(* PLC project KA107__GPA2.project, Prosoft-Systems Ltd. Astra.IDE Astra.IDE_V1.7.2.1 *)
(* stored: creationDateTime 2025-08-26T12:04:32.1909898, modificationDateTime 2025-08-26T12:03:09.7987139 *)

///
///Назначение: 		готовности к пуску
///Автор: 				Korsuntsev/Chekmarev 20/02/2025
///Версия: 			00.00.02
///Проект: 			КА107
{attribute 'qualified_only' := ''}
{attribute 'strict' := ''}
{attribute 'symbol' := 'none'}
TYPE ENUM_ReadyToStart :
(
	/// Готовность отключена
	OFF := 0,
	/// Готовность к ХП
	HP := 1,
	/// Готовность к КПК
	KPK := 2,
	/// Готовность к АПК
	APK := 3
) USINT;
END_TYPE

PROGRAM DIAGN

                    REDUNDANCY();
UCP1_A1_1();
UCP1_A2_1();
UE1_A1_1();

                  

ACTION UE1_A1_1:
                        PsDiagn.PROXY_ST_XX_X1X(MODULE := UE1_A1_ST1, DATA := MODULE_UE1_A1_ST1);
PsDiagn.PROXY_PP_00_XXX(MODULE := UE1_A1_PP1, DATA := MODULE_UE1_A1_PP1);
PsDiagn.PROXY_AI_16_011(MODULE := UE1_A1_DI1, DATA := MODULE_UE1_A1_DI1);
PsDiagn.PROXY_AI_16_011(MODULE := UE1_A1_DI2, DATA := MODULE_UE1_A1_DI2);
PsDiagn.PROXY_AI_16_011(MODULE := UE1_A1_DI3, DATA := MODULE_UE1_A1_DI3);
PsDiagn.PROXY_DI_32_011(MODULE := UE1_A1_DI4, DATA := MODULE_UE1_A1_DI4);
PsDiagn.PROXY_DI_32_011(MODULE := UE1_A1_DI5, DATA := MODULE_UE1_A1_DI5);
PsDiagn.PROXY_DO_32_012(MODULE := UE1_A1_DO1, DATA := MODULE_UE1_A1_DO1);
PsDiagn.PROXY_DI_32_011(MODULE := UE1_A1_DI6, DATA := MODULE_UE1_A1_DI6);
PsDiagn.PROXY_DO_32_012(MODULE := UE1_A1_DO2, DATA := MODULE_UE1_A1_DO2);
PsDiagn.PROXY_DI_32_011(MODULE := UE1_A1_DI7, DATA := MODULE_UE1_A1_DI7);
PsDiagn.PROXY_ST_XX_X2X(MODULE := UE1_A1_ST2, DATA := MODULE_UE1_A1_ST2);

                      
END_ACTION

ACTION UCP1_A2_1:
                        PsDiagn.PROXY_ST_XX_X1X(MODULE := UCP1_A2_ST1, DATA := MODULE_UCP1_A2_ST1);
PsDiagn.PROXY_PP_00_XXX(MODULE := UCP1_A2_PP1, DATA := MODULE_UCP1_A2_PP1);
PsDiagn.PROXY_AO_08_031(MODULE := UCP1_A2_AO1, DATA := MODULE_UCP1_A2_AO1);
PsDiagn.PROXY_AI_16_011(MODULE := UCP1_A2_DI1, DATA := MODULE_UCP1_A2_DI1);
PsDiagn.PROXY_AI_16_011(MODULE := UCP1_A2_DI2, DATA := MODULE_UCP1_A2_DI2);
PsDiagn.PROXY_DI_32_011(MODULE := UCP1_A2_DI3, DATA := MODULE_UCP1_A2_DI3);
PsDiagn.PROXY_DO_32_012(MODULE := UCP1_A2_DO1, DATA := MODULE_UCP1_A2_DO1);
PsDiagn.PROXY_DI_32_011(MODULE := UCP1_A2_DI4, DATA := MODULE_UCP1_A2_DI4);
PsDiagn.PROXY_ST_XX_X2X(MODULE := UCP1_A2_ST2, DATA := MODULE_UCP1_A2_ST2);

                      
END_ACTION

ACTION REDUNDANCY:
                        //Активный ПЛК
IS_ACTIVE := TRUE;

//ПЛК А
IS_CPU_A := TRUE;

//ПЛК В
IS_CPU_B := FALSE;


                      
END_ACTION

ACTION UCP1_A1_1:
                        PsDiagn.PROXY_ST_XX_X1X(MODULE := UCP1_A1_ST1, DATA := MODULE_UCP1_A1_ST1);
PsDiagn.PROXY_PP_00_XXX(MODULE := UCP1_A1_PP1, DATA := MODULE_UCP1_A1_PP1);
PsDiagn.GET_CPU_INFO_R500(REGULBUS_HW := Regul_Bus_OS.HwError, SYNC_OK := TRUE, HW := UCP1_A1_CU1.HwError, PF := FALSE, INFO => MODULE_UCP1_A1_CU1);
PsDiagn.PROXY_DA_03_021_L_FRQ(MODULE := UCP1_A1_FI1, DATA := MODULE_UCP1_A1_FI1);
PsDiagn.PROXY_DA_03_021_L_FRQ(MODULE := UCP1_A1_FI2, DATA := MODULE_UCP1_A1_FI2);
PsDiagn.PROXY_AI_08_052(MODULE := UCP1_A1_AI1, DATA := MODULE_UCP1_A1_AI1);
PsDiagn.PROXY_AI_08_052(MODULE := UCP1_A1_AI2, DATA := MODULE_UCP1_A1_AI2);
PsDiagn.PROXY_AI_08_052(MODULE := UCP1_A1_AI3, DATA := MODULE_UCP1_A1_AI3);
PsDiagn.PROXY_AI_08_031(MODULE := UCP1_A1_AI4, DATA := MODULE_UCP1_A1_AI4);
PsDiagn.PROXY_AI_08_031(MODULE := UCP1_A1_AI5, DATA := MODULE_UCP1_A1_AI5);
PsDiagn.PROXY_AI_08_031(MODULE := UCP1_A1_AI6, DATA := MODULE_UCP1_A1_AI6);
PsDiagn.PROXY_AI_08_031(MODULE := UCP1_A1_AI7, DATA := MODULE_UCP1_A1_AI7);
PsDiagn.PROXY_ST_XX_X2X(MODULE := UCP1_A1_ST2, DATA := MODULE_UCP1_A1_ST2);

                      
END_ACTION
END_PROGRAM

FUNCTION FC_PrepareShutdown : DWORD
VAR_IN_OUT
	EventPrm: Component_Manager.EVTPARAM_CmpMgr_Shutdown;
END_VAR
VAR
END_VAR

                    IS_ACTIVE := FALSE;
IS_CPU_A := FALSE;
IS_CPU_B := FALSE;

                  
END_FUNCTION

FUNCTION FC_StopDone : DWORD
VAR_IN_OUT
	EventPrm: CmpApp.EVTPARAM_CmpAppStop;
END_VAR
VAR
END_VAR

                    IS_ACTIVE := FALSE;
IS_CPU_A := FALSE;
IS_CPU_B := FALSE;

                  
END_FUNCTION

FUNCTION FC_Exception : DWORD
VAR_IN_OUT
	EventPrm: CmpApp.EVTPARAM_CmpAppException;
END_VAR
VAR
END_VAR

                    IS_ACTIVE := FALSE;
IS_CPU_A := FALSE;
IS_CPU_B := FALSE;

                  
END_FUNCTION

{attribute 'linkalways' := ''}
PROGRAM PRG_9d6fa412_87bb_44d3_b4af_3b2a0d18f6a8

                    {IF defined (pou: SETPOINTS_PRG_STORE_060ed6ea_c6b5_480d_b15e_3bc8654c83ea)}
SETPOINTS_PRG_STORE_060ed6ea_c6b5_480d_b15e_3bc8654c83ea();
{END_IF}
                  
END_PROGRAM

{attribute 'linkalways' := ''}
PROGRAM PRG_b5ed8c35_93f2_4693_9ede_6cbb2df9f327

                    {IF defined (pou: SETPOINTS_PRG_RESTORE_926b34b1_d125_4ae4_9712_933a3ae333bd)}
SETPOINTS_PRG_RESTORE_926b34b1_d125_4ae4_9712_933a3ae333bd();
{END_IF}
                  
END_PROGRAM

PROGRAM PRG_base
VAR
 	//Время выполнения программы
	result_time:ULINT;
	/// Признак первого вызова программы
	init: BOOL := TRUE;
END_VAR
VAR_TEMP
	start_time:ULINT;
	end_time:ULINT;
END_VAR

                    start_time:= PsTimeGetUtcTimeNs(); // Время начала выполнения
//==============================================================================================

IF init THEN
	fun_init();
	init := FALSE;
END_IF

//Кнопки
btn_update();

// Настройки
tunpar_update();

// Таймеры
tmr_update();

// ИМ-ы
// Конфигуратор
am_update();
// Создан вручную
am_update_base();

//Алгоритм
ALG_base();				//Алгоритм

aggregation_am();

// Формирование тестовых сигналов
test.Saw_Slow();
test.Sin_Slow();

//==============================================================================================
end_time:=PsTimeGetUtcTimeNs() ;  // конец
result_time:=end_time-start_time;  // время выполнения фрагмента кода
                  
END_PROGRAM

PROGRAM PRG_fast
VAR
 	//Время выполнения программы
	result_time:ULINT;
END_VAR
VAR_TEMP
	start_time:ULINT;
	end_time:ULINT;
END_VAR

                    start_time:=PsTimeGetUtcTimeNs(); // Время начала выполнения
//==============================================================================================

////// Временно здесь
//{warning ' Убрать на новой версии макроса '}
//aipar.common.sim_aggregated	:= FALSE;
//aopar.common.sim_aggregated	:= FALSE;
//dipar.common.sim_aggregated	:= FALSE;
//dopar.common.sim_aggregated	:= FALSE;
/////////////

// Сброс переменных VAR_STAT
// По входам / выходам
reset_io_var_stat();
// По сигнализациям
reset_alarm_var_stat();
// По ИМам
reset_am_var_stat();

// Ввод
	aipar_update(cycle := cycle_time_fast);		//Вызов обработки всех экземпляров AI быстрого цикла
	dipar_update();								//Вызов обработки всех экземпляров DI быстрого цикла
	
	MODULE_UCP1_A1_AI6.T_JUNCTION := aipar.Tcool.value; // компенсация холодного спая
	MODULE_UCP1_A1_AI7.T_JUNCTION := aipar.Tcool.value; // компенсация холодного спая
//---------------------------------------------------------------------------------------------

// Расчётные параметры
	acpar_handler.handler(cycle := cycle_time_fast);
	
	acpar_update(); 							//Обработка расчётных параметров (Формирование уставок)
//---------------------------------------------------------------------------------------------	

// Сигнализации
	Alarm_link(); //Подготовка данных и вызов обработчиков сигнализаций
//Агрегация сигнализаций (все сигнализации должны быть вызваны к этому моменту)
	aggregation_alarms();
//---------------------------------------------------------------------------------------------	

// Топливный регулятор
	FR_link();
	AS_Link();

// Быстрые ИМ-ы
	ALG_D_AM_fast();
	// Создан вручную
	am_update_fast();
	// аналоговые
	// Конфигуратор
	ama_update();

//Сигналы контроллера
	ALG_PLC();

// Вывод
	aopar_update(); 							//Вызов обработки всех экземпляров AO быстрого цикла
	dopar_update(); 							//Вызов обработки всех экземпляров DO быстрого цикла
//---------------------------------------------------------------------------------------------	
// IEC 104

// Формирование тестовых сигналов
	test.Saw_Fast();
// IEC-104
	IEC104_update();

//==============================================================================================
end_time:=PsTimeGetUtcTimeNs() ;  // конец
result_time:=end_time-start_time;  // время выполнения фрагмента кода

                  
END_PROGRAM

PROGRAM PRG_slow

                    handleMotoClock();
alg.sh_cntrl := ShCntrl();
                  
END_PROGRAM

{region INFO}
(*
 Назначение: Используется для вызова предупредительных и ограничительных сигнализаций
 Автор:  /Andrey/ 24.06.2025 16:50:31
 Версия: v00.00.22
 Проект: KA107__GPA2
*)
{endregion}
FUNCTION alr_update : BOOL
VAR_INPUT
END_VAR

                    //==========================================================================

//==========================================================================
//Подсистема: Внешние источники
//--------------------------------------------------------------------------
//Кнопка ЭАО на ПРУ нажата сигнал 1 (НР)
alr.EAO_PRU_1(
in     := dipar.EAO_PRU_1.value,
cmd_on := TRUE, cmd_off  := FALSE);
//--------------------------------------------------------------------------

//Кнопка ЭАО на ПРУ нажата сигнал 2 (НЗ)
alr.EAO_PRU_2(
in     := dipar.EAO_PRU_2.value,
cmd_on := TRUE, cmd_off  := FALSE);
//--------------------------------------------------------------------------

//Кнопка ЭАО на ПРУ нажата сигнал 3 (НЗ)
alr.EAO_PRU_3(
in     := dipar.EAO_PRU_3.value,
cmd_on := TRUE, cmd_off  := FALSE);
//--------------------------------------------------------------------------

//Нет связи с ПРУ
alr.PRU_noLink(
in     := NOT PRU.Link,
cmd_on := TRUE, cmd_off  := FALSE);
//--------------------------------------------------------------------------

//==========================================================================

//==========================================================================
//Подсистема: Блок двигателя
//--------------------------------------------------------------------------
//Загазованность контейнеров выше нормы
alr.Zagaz_OD_Pv(
in     := dipar.Zagaz_OD_Pv.value,
cmd_on := TRUE, cmd_off  := FALSE);
//--------------------------------------------------------------------------

//Повышенная вибрация двигателя
alr.Vs_D_Pv(
in     := dipar.Vs_D_Pv.value,
cmd_on := TRUE, cmd_off  := FALSE);
//--------------------------------------------------------------------------

//Повыш. Вибрация ТК
alr.Vstk_H(
in     := aipar.Vstk.setpoint.H,
cmd_on := TRUE, cmd_off  := FALSE);
//--------------------------------------------------------------------------

//Повыш. Вибрация СТ
alr.Vsst_H(
in     := aipar.Vsst.setpoint.H,
cmd_on := TRUE, cmd_off  := FALSE);
//--------------------------------------------------------------------------

//Сигнализатор обледенения
alr.Ace_alr(
in     := dipar.Ace_alr.value,
cmd_on := TRUE, cmd_off  := FALSE);
//--------------------------------------------------------------------------

//КПВ не открыты на пуске
alr.KPV_nOpen(
in     := NOT ( dipar.KPV2_ON.value AND dipar.KPV3_ON.value AND dipar.KPV4_ON.value AND dipar.KPV1_ON.value AND dipar.KPV5_ON.value ),
cmd_on := acpar.Ntk.value > 2000 AND acpar.Ntk.value < 4500 AND alg.start, cmd_off  := acpar.Ntk.value > 4500 OR alg.AO);
//--------------------------------------------------------------------------

//КПВ234 не открыты
alr.KPV234_nOpen(
in     := NOT ( dipar.KPV2_ON.value AND dipar.KPV3_ON.value AND dipar.KPV4_ON.value ),
cmd_on := NOss.cmd_KPV234_On OR NObs.cmd_KPV234_On OR AOss.cmd_KPV234_On OR AObs.cmd_KPV234_On, cmd_off  := acpar.Ntk.value < 2000);
//--------------------------------------------------------------------------

//Повыш. Обороты СТ > 8500 об/мин
alr.Nst_H(
in     := acpar.Nst.setpoint.H,
cmd_on := TRUE, cmd_off  := FALSE);
//--------------------------------------------------------------------------

//Высокая скорость изменения оборотов 1-ого канала ТК
alr.Ntk_1_OV(
in     := acpar_handler.handler.nTKcalc.fltUcv[1],
cmd_on := TRUE, cmd_off  := FALSE);
//--------------------------------------------------------------------------

//Высокая скорость изменения оборотов 2-ого канала ТК
alr.Ntk_2_OV(
in     := acpar_handler.handler.nTKcalc.fltUcv[2],
cmd_on := TRUE, cmd_off  := FALSE);
//--------------------------------------------------------------------------

//Значения оборотов 1-ого канала ТК не в диапазоне
alr.Ntk_1_UV(
in     := acpar_handler.handler.nTKcalc.flt[1],
cmd_on := TRUE, cmd_off  := FALSE);
//--------------------------------------------------------------------------

//Значения оборотов 2-ого канала ТК не в диапазоне
alr.Ntk_2_UV(
in     := acpar_handler.handler.nTKcalc.flt[2],
cmd_on := TRUE, cmd_off  := FALSE);
//--------------------------------------------------------------------------

//Значения оборотов 1-ого канала СТ не в диапазоне
alr.Nst_1_UV(
in     := acpar_handler.handler.nSTcalc.flt[1],
cmd_on := TRUE, cmd_off  := FALSE);
//--------------------------------------------------------------------------

//Значения оборотов 2-ого канала СТ не в диапазоне
alr.Nst_2_UV(
in     := acpar_handler.handler.nSTcalc.flt[2],
cmd_on := TRUE, cmd_off  := FALSE);
//--------------------------------------------------------------------------

//Высокая скорость изменения оборотов 1-ого канала СТ
alr.Nst_1_OV(
in     := acpar_handler.handler.nSTcalc.fltUcv[1],
cmd_on := TRUE, cmd_off  := FALSE);
//--------------------------------------------------------------------------

//Высокая скорость изменения оборотов 2-ого канала СТ
alr.Nst_2_OV(
in     := acpar_handler.handler.nSTcalc.fltUcv[2],
cmd_on := TRUE, cmd_off  := FALSE);
//--------------------------------------------------------------------------

//Повыш. Температура газа на входе СТ
alr.Tg_inST_H(
in     := acpar.Tg_inST.setpoint.H,
cmd_on := TRUE, cmd_off  := FALSE);
//--------------------------------------------------------------------------

//Нет сигнала: ТРК: готовность
alr.N_TRKready(
in     := NOT dipar.TRKready.value,
cmd_on := TRUE, cmd_off  := FALSE);
//--------------------------------------------------------------------------

//ТРК: авария
alr.TRKalr(
in     := dipar.TRKalr.value,
cmd_on := TRUE, cmd_off  := FALSE);
//--------------------------------------------------------------------------

//Контроль САУ не пройден
alr.nCheckSAU(
in     := check.tmrCancelPrm.Q,
cmd_on := TRUE, cmd_off  := FALSE);
//--------------------------------------------------------------------------

//Неисправность БЗА
alr.BZA_flt(
in     := NOT dipar.BZA_ready_1.value OR NOT dipar.BZA_ready_2.value,
cmd_on := tch.GTDWork.value, cmd_off  := NOT tch.GTDWork.value);
//--------------------------------------------------------------------------

//==========================================================================

//==========================================================================
//Подсистема: Маслосистема двигателя
//--------------------------------------------------------------------------
//Пониж. Температура масла на входе двигателя
alr.Tm_inD_L(
in     := aipar.Tm_inD.setpoint.L,
cmd_on := TRUE, cmd_off  := FALSE);
//--------------------------------------------------------------------------

//Уровень масла в МБД+Н минимальный
alr.Lm_MB_Pn(
in     := dipar.Lm_MB_Pn.value,
cmd_on := TRUE, cmd_off  := FALSE);
//--------------------------------------------------------------------------

//==========================================================================

//==========================================================================
//Подсистема: Воздушный стартер
//--------------------------------------------------------------------------
//==========================================================================

//==========================================================================
//Подсистема: Аппарат воздушного охлаждения масла двигателя
//--------------------------------------------------------------------------
//Повыш. Температура масла на выходе АВОМД
alr.Tm_outAVOM_H(
in     := aipar.Tm_outAVOM.setpoint.H,
cmd_on := TRUE, cmd_off  := FALSE);
//--------------------------------------------------------------------------

//Неисправность вентилятора 1 АВОМД
alr.Vn1_AVOM_flt(
in     := am.Vn1_AVOM.flt,
cmd_on := TRUE, cmd_off  := FALSE);
//--------------------------------------------------------------------------

//Неисправность вентилятора 2 АВОМД
alr.Vn2_AVOM_flt(
in     := am.Vn2_AVOM.flt,
cmd_on := TRUE, cmd_off  := FALSE);
//--------------------------------------------------------------------------

//Неисправность вентилятора 3 АВОМД
alr.Vn3_AVOM_flt(
in     := am.Vn3_AVOM.flt,
cmd_on := TRUE, cmd_off  := FALSE);
//--------------------------------------------------------------------------

//Неисправность вентилятора 4 АВОМД
alr.Vn4_AVOM_flt(
in     := am.Vn4_AVOM.flt,
cmd_on := TRUE, cmd_off  := FALSE);
//--------------------------------------------------------------------------

//==========================================================================

//==========================================================================
//Подсистема: Блок топливного газа
//--------------------------------------------------------------------------
//Пониж. Давление топливного газа перед ТРК
alr.Ptg_inTRK_L(
in     := aipar.Ptg_inTRK.setpoint.L,
cmd_on := alg.sh_TG, cmd_off  := NOT alg.sh_TG);
//--------------------------------------------------------------------------

//Повыш. Давление топливного газа перед ТРК
alr.Ptg_inTRK_H(
in     := aipar.Ptg_inTRK.setpoint.H,
cmd_on := true, cmd_off  := false);
//--------------------------------------------------------------------------

//Давление газа перед дозатором газа Предупредительное
alr.Ptg_inDG_Pn(
in     := dipar.Ptg_inDG_Pn.value,
cmd_on := alg.sh_TG, cmd_off  := NOT alg.sh_TG);
//--------------------------------------------------------------------------

//==========================================================================

//==========================================================================
//Подсистема: Блок пускового газа
//--------------------------------------------------------------------------
//==========================================================================

//==========================================================================
//Подсистема: Противообледенительная система и воздухоочистное устройство
//--------------------------------------------------------------------------
//Перепад на сетке ВОУ
alr.Exh_VOU(
in     := dipar.Exh_VOU.value,
cmd_on := TRUE, cmd_off  := FALSE);
//--------------------------------------------------------------------------

//==========================================================================

//==========================================================================
//Подсистема: Компрессорная установка/блок нагнетателя
//--------------------------------------------------------------------------
//Опасность помпажа нагнетателя
alr.AS_Pv(
in     := s_tunpar.ASprot.emergOpenBypass,
cmd_on := TRUE, cmd_off  := FALSE);
//--------------------------------------------------------------------------

//Пониж. Перепад давления “масло-газ”
alr.dPmg_L(
in     := aipar.dPmg.setpoint.L,
cmd_on := alg.sh_dPmg, cmd_off  := NOT alg.sh_dPmg);
//--------------------------------------------------------------------------

//Уровень масла в МБУпл минимальный
alr.Lm_MBU_Pn(
in     := dipar.Lm_MBU_Pn.value,
cmd_on := TRUE, cmd_off  := FALSE);
//--------------------------------------------------------------------------

//Повыш. Температура упорного подшипника Н
alr.Tup_N_H(
in     := aipar.Tup_N.setpoint.H,
cmd_on := TRUE, cmd_off  := FALSE);
//--------------------------------------------------------------------------

//Повыш. Температура опорного подшипника №1 Н
alr.Top_N_1_H(
in     := aipar.Top_N_1.setpoint.H,
cmd_on := TRUE, cmd_off  := FALSE);
//--------------------------------------------------------------------------

//Повыш. Температура опорного подшипника №2 Н
alr.Top_N_2_H(
in     := aipar.Top_N_2.setpoint.H,
cmd_on := TRUE, cmd_off  := FALSE);
//--------------------------------------------------------------------------

//Давление масла смазки Н предупредительная
alr.Pm_N_Pn(
in     := dipar.Pm_N_Pn.value,
cmd_on := NOT alg.V_000, cmd_off  := alg.V_000);
//--------------------------------------------------------------------------

//==========================================================================

//==========================================================================
//Подсистема: Блок управления
//--------------------------------------------------------------------------
//Нет сигнала: Предохранитель UCP1-XTFU1:1 питания модулей AO исправен
alr.N_Fuse_AO_UCP1(
in     := NOT dipar.Fuse_AO_UCP1.value,
cmd_on := TRUE, cmd_off  := FALSE);
//--------------------------------------------------------------------------

//Нет сигнала: Предохранитель UCP1-XTFU1:2 питания модулей DO исправен
alr.N_Fuse_DO_UCP1(
in     := NOT dipar.Fuse_DO_UCP1.value,
cmd_on := TRUE, cmd_off  := FALSE);
//--------------------------------------------------------------------------

//Нет сигнала: Предохранитель UCP1--XTFU6:1 питания датчиков температуры и влажности
alr.N_Fuse_Air_UCP1(
in     := NOT dipar.Fuse_Air_UCP1.value,
cmd_on := TRUE, cmd_off  := FALSE);
//--------------------------------------------------------------------------

//Нет сигнала: Предохранитель UE1-XTFU1:2 питания модулей DO исправен
alr.N_Fuse_DO_UE1(
in     := NOT dipar.Fuse_DO_UE1.value,
cmd_on := TRUE, cmd_off  := FALSE);
//--------------------------------------------------------------------------

//Перегрузка фильтра EV1 (Осн.)
alr.EV1(
in     := dipar.EV1.value,
cmd_on := TRUE, cmd_off  := FALSE);
//--------------------------------------------------------------------------

//Перегрузка фильтра EV2 (Рез.)
alr.EV2(
in     := dipar.EV2.value,
cmd_on := TRUE, cmd_off  := FALSE);
//--------------------------------------------------------------------------

//Нет сигнала: Контроль основного ввода питания (-KV1)
alr.N_U_main(
in     := NOT dipar.U_main.value,
cmd_on := TRUE, cmd_off  := FALSE);
//--------------------------------------------------------------------------

//Нет сигнала: Контроль резервного ввода питания (-KV2)
alr.N_U_res(
in     := NOT dipar.U_res.value,
cmd_on := TRUE, cmd_off  := FALSE);
//--------------------------------------------------------------------------

//Контроль замыкания на землю питания PLC
alr.U_G_PLC(
in     := dipar.U_G_PLC.value,
cmd_on := TRUE, cmd_off  := FALSE);
//--------------------------------------------------------------------------

//Контроль замыкания на землю питания AI
alr.U_G_AI(
in     := dipar.U_G_AI.value,
cmd_on := TRUE, cmd_off  := FALSE);
//--------------------------------------------------------------------------

//Контроль замыкания на землю питания DI
alr.U_G_DI(
in     := dipar.U_G_DI.value,
cmd_on := TRUE, cmd_off  := FALSE);
//--------------------------------------------------------------------------

//Контроль замыкания на землю питания БИЗ
alr.U_G_BIZ(
in     := dipar.U_G_BIZ.value,
cmd_on := TRUE, cmd_off  := FALSE);
//--------------------------------------------------------------------------

//Нет сигнала: Контроль -AG1
alr.N_AG1(
in     := NOT dipar.AG1.value,
cmd_on := TRUE, cmd_off  := FALSE);
//--------------------------------------------------------------------------

//Нет сигнала: Контроль -AG2
alr.N_AG2(
in     := NOT dipar.AG2.value,
cmd_on := TRUE, cmd_off  := FALSE);
//--------------------------------------------------------------------------

//Нет сигнала: Контроль -AG3
alr.N_AG3(
in     := NOT dipar.AG3.value,
cmd_on := TRUE, cmd_off  := FALSE);
//--------------------------------------------------------------------------

//Нет сигнала: Контроль -AG4
alr.N_AG4(
in     := NOT dipar.AG4.value,
cmd_on := TRUE, cmd_off  := FALSE);
//--------------------------------------------------------------------------

//Нет сигнала: Контроль -AG9
alr.N_AG9(
in     := NOT dipar.AG9.value,
cmd_on := TRUE, cmd_off  := FALSE);
//--------------------------------------------------------------------------

//Нет сигнала: Контроль -AG10
alr.N_AG10(
in     := NOT dipar.AG10.value,
cmd_on := TRUE, cmd_off  := FALSE);
//--------------------------------------------------------------------------

//Нет сигнала: Контроль -AG15
alr.N_AG15(
in     := NOT dipar.AG15.value,
cmd_on := TRUE, cmd_off  := FALSE);
//--------------------------------------------------------------------------

//Нет сигнала: Контроль -AG16
alr.N_AG16(
in     := NOT dipar.AG16.value,
cmd_on := TRUE, cmd_off  := FALSE);
//--------------------------------------------------------------------------

//Нет сигнала: Контроль -AG5
alr.N_AG5(
in     := NOT dipar.AG5.value,
cmd_on := TRUE, cmd_off  := FALSE);
//--------------------------------------------------------------------------

//Нет сигнала: Контроль -AG6
alr.N_AG6(
in     := NOT dipar.AG6.value,
cmd_on := TRUE, cmd_off  := FALSE);
//--------------------------------------------------------------------------

//Нет сигнала: Контроль -AG8
alr.N_AG8(
in     := NOT dipar.AG8.value,
cmd_on := TRUE, cmd_off  := FALSE);
//--------------------------------------------------------------------------

//Нет сигнала: Контроль -AG17
alr.N_AG17(
in     := NOT dipar.AG17.value,
cmd_on := TRUE, cmd_off  := FALSE);
//--------------------------------------------------------------------------

//Нет сигнала: Контроль -AG18
alr.N_AG18(
in     := NOT dipar.AG18.value,
cmd_on := TRUE, cmd_off  := FALSE);
//--------------------------------------------------------------------------

//Нет сигнала: Контроль питания ПРУ
alr.N_U_PRU(
in     := NOT dipar.U_PRU.value,
cmd_on := TRUE, cmd_off  := FALSE);
//--------------------------------------------------------------------------

//Нет сигнала: Контроль питания ТРК осн.
alr.N_Utrk_main(
in     := NOT dipar.Utrk_main.value,
cmd_on := TRUE, cmd_off  := FALSE);
//--------------------------------------------------------------------------

//Контроль замыкания на землю питания ИМ
alr.U_G_AM(
in     := dipar.U_G_AM.value,
cmd_on := TRUE, cmd_off  := FALSE);
//--------------------------------------------------------------------------

//Нет сигнала: Контроль питания AI
alr.N_U_AI(
in     := NOT dipar.U_AI.value,
cmd_on := TRUE, cmd_off  := FALSE);
//--------------------------------------------------------------------------

//Нет сигнала: Контроль питания DI
alr.N_U_DI(
in     := NOT dipar.U_DI.value,
cmd_on := TRUE, cmd_off  := FALSE);
//--------------------------------------------------------------------------

//Нет сигнала: Контроль питания БИЗ
alr.N_U_BIZ(
in     := NOT dipar.U_BIZ.value,
cmd_on := TRUE, cmd_off  := FALSE);
//--------------------------------------------------------------------------

//Нет сигнала: Контроль питания ИМ
alr.N_U_AM(
in     := NOT dipar.U_AM.value,
cmd_on := TRUE, cmd_off  := FALSE);
//--------------------------------------------------------------------------

//Нет сигнала: Контроль питания аппаратуры вибрации, =24 В
alr.N_Uvs_24(
in     := NOT dipar.Uvs_24.value,
cmd_on := TRUE, cmd_off  := FALSE);
//--------------------------------------------------------------------------

//Нет сигнала: Контроль питания дополнительного оборудования, =24В
alr.N_Uother_24(
in     := NOT dipar.Uother_24.value,
cmd_on := TRUE, cmd_off  := FALSE);
//--------------------------------------------------------------------------

//Нет сигнала: Контроль питания ИМ2
alr.N_U_AM2(
in     := NOT dipar.U_AM2.value,
cmd_on := TRUE, cmd_off  := FALSE);
//--------------------------------------------------------------------------

//Нет сигнала: Контроль питания ТРК рез.
alr.N_Utrk_res(
in     := NOT dipar.Utrk_res.value,
cmd_on := TRUE, cmd_off  := FALSE);
//--------------------------------------------------------------------------

//БЭО. Перегрузка фильтра EV3 (Осн. БЭО)
alr.EV3(
in     := dipar.EV3.value,
cmd_on := TRUE, cmd_off  := FALSE);
//--------------------------------------------------------------------------

//БЭО. Перегрузка фильтра EV4 (Рез. БЭО)
alr.EV4(
in     := dipar.EV4.value,
cmd_on := TRUE, cmd_off  := FALSE);
//--------------------------------------------------------------------------

//Нет сигнала: БЭО. Контроль основного ввода питания БЭО (-KV3)
alr.N_Ubeo_main(
in     := NOT dipar.Ubeo_main.value,
cmd_on := TRUE, cmd_off  := FALSE);
//--------------------------------------------------------------------------

//Нет сигнала: БЭО. Контроль резервного ввода питания БЭО (-KV4)
alr.N_Ubeo_res(
in     := NOT dipar.Ubeo_res.value,
cmd_on := TRUE, cmd_off  := FALSE);
//--------------------------------------------------------------------------

//Нет сигнала: БЭО. Контроль -AG11
alr.N_AG11(
in     := NOT dipar.AG11.value,
cmd_on := TRUE, cmd_off  := FALSE);
//--------------------------------------------------------------------------

//Нет сигнала: БЭО. Контроль -AG12
alr.N_AG12(
in     := NOT dipar.AG12.value,
cmd_on := TRUE, cmd_off  := FALSE);
//--------------------------------------------------------------------------

//БЭО. Контроль замыкания на землю питания БЭО (-KR5)
alr.U_G_KR5(
in     := dipar.U_G_KR5.value,
cmd_on := TRUE, cmd_off  := FALSE);
//--------------------------------------------------------------------------

//Нет сигнала: БЭО. Контроль питания кн. ЭАО
alr.N_U_KEAO(
in     := NOT dipar.U_KEAO.value,
cmd_on := TRUE, cmd_off  := FALSE);
//--------------------------------------------------------------------------

//Нет сигнала: БЭО. Контроль питания БЭО
alr.N_U_BEO(
in     := NOT dipar.U_BEO.value,
cmd_on := TRUE, cmd_off  := FALSE);
//--------------------------------------------------------------------------

//Нет сигнала: БЭО. Контроль питания БЗА
alr.N_U_BZA(
in     := NOT dipar.U_BZA.value,
cmd_on := TRUE, cmd_off  := FALSE);
//--------------------------------------------------------------------------

//Ошибка -AUO1
alr.Err_AUO1(
in     := dipar.Err_AUO1.value,
cmd_on := TRUE, cmd_off  := FALSE);
//--------------------------------------------------------------------------

//==========================================================================

//==========================================================================
//Подсистема: Газовая обвязка
//--------------------------------------------------------------------------
//==========================================================================

//==========================================================================
//Подсистема: Контроль защит
//--------------------------------------------------------------------------
//Одна или более защит не взведены
alr.shCntrl(
in     := NOT alg.sh_cntrl,
cmd_on := TRUE, cmd_off  := FALSE);
//--------------------------------------------------------------------------

                  
END_FUNCTION

{region INFO}
(*
 Назначение: Используется для вызова аварийных сигнализаций
 Автор:  /Andrey/ 24.06.2025 16:50:31
 Версия: v00.00.22
 Проект: KA107__GPA2
*)
{endregion}
FUNCTION crs_update : BOOL
VAR_INPUT
END_VAR

                    //==========================================================================

//==========================================================================
//Подсистема: Внешние источники
//--------------------------------------------------------------------------
//АОсс: АОсс от оператора
crs.btn_AOss(
in        := btn.AOss.out,
brk       := FALSE,
cmd_on    := TRUE, cmd_off  := FALSE);
//--------------------------------------------------------------------------

//АОбс: АОбс от оператора
crs.btn_AObs(
in        := btn.AObs.out,
brk       := FALSE,
cmd_on    := TRUE, cmd_off  := FALSE);
//--------------------------------------------------------------------------

//АОсс: АОсс по технологическим условиям
crs.AOss_tech(
in        := alg.AOss_tech,
brk       := FALSE,
cmd_on    := TRUE, cmd_off  := FALSE);
//--------------------------------------------------------------------------

//АОбс: АОбс по технологическим условиям
crs.AObs_tech(
in        := alg.AOss_tech,
brk       := FALSE,
cmd_on    := TRUE, cmd_off  := FALSE);
//--------------------------------------------------------------------------

//АОсс: Кнопка АО на ПРУ
crs.AO_PRU(
in        := dipar.AO_PRU_1.value OR dipar.AO_PRU_2.value,
brk       := dipar.AO_PRU_1.flt OR dipar.AO_PRU_2.flt,
cmd_on    := TRUE, cmd_off  := FALSE);
//--------------------------------------------------------------------------

//АОсс: АО от кнопки "АО" блока автоматики ГПА
crs.AO_BA(
in        := dipar.AO_BA.value,
brk       := dipar.AO_BA.flt,
cmd_on    := TRUE, cmd_off  := FALSE);
//--------------------------------------------------------------------------

//АОсс: БЭАО сработал
crs.BEAO(
in        := dipar.BEAO.value,
brk       := dipar.BEAO.flt,
cmd_on    := TRUE, cmd_off  := FALSE);
//--------------------------------------------------------------------------

//==========================================================================

//==========================================================================
//Подсистема: Блок двигателя
//--------------------------------------------------------------------------
//АОбс: Самопроизвольное закрытие СК
crs.Causeless_SK(
in        := NOT dipar.SK_ON.value,
brk       := dipar.SK_ON.flt,
cmd_on    := FuelReg.fReg.isFire, cmd_off  := NOT am.SK.on);
//--------------------------------------------------------------------------

//АОсс: Помпаж двигателя
crs.SurgeD(
in        := dipar.SurgeD.value,
brk       := dipar.SurgeD.flt,
cmd_on    := TRUE, cmd_off  := FALSE);
//--------------------------------------------------------------------------

//АОсс: Опасная вибрация двигателя
crs.Vs_D_Av(
in        := dipar.Vs_D_Av.value,
brk       := dipar.Vs_D_Av.flt,
cmd_on    := TRUE, cmd_off  := FALSE);
//--------------------------------------------------------------------------

//АОбс: Авар.-выс. Вибрация ТК
crs.Vstk_HH(
in        := aipar.Vstk.setpoint.HH,
brk       := aipar.Vstk.flt,
cmd_on    := TRUE, cmd_off  := FALSE);
//--------------------------------------------------------------------------

//АОсс: Авар.-выс. Вибрация СТ
crs.Vsst_HH(
in        := aipar.Vsst.setpoint.HH,
brk       := aipar.Vsst.flt,
cmd_on    := TRUE, cmd_off  := FALSE);
//--------------------------------------------------------------------------

//АОбс: КПВ234 не закрыты
crs.KPV234_wOpen(
in        := NOT ( dipar.KPV2_off.value AND dipar.KPV3_off.value AND dipar.KPV4_off.value ),
brk       := dipar.KPV2_off.flt OR dipar.KPV3_off.flt OR dipar.KPV4_off.flt,
cmd_on    := alg.KPV234_wOpen, cmd_off  := NOT alg.KPV234_wOpen);
//--------------------------------------------------------------------------

//АОбс: КПВ15 не закрыты
crs.KPV15_wOpen(
in        := NOT ( dipar.KPV1_off.value AND dipar.KPV5_off.value ),
brk       := dipar.KPV1_off.flt OR dipar.KPV5_off.flt,
cmd_on    := alg.KPV15_wOpen, cmd_off  := NOT alg.KPV15_wOpen);
//--------------------------------------------------------------------------

//АОбс: КПВ15 не открыты
crs.KPV15_nOpen(
in        := NOT ( dipar.KPV1_ON.value AND dipar.KPV5_ON.value ),
brk       := dipar.KPV1_ON.flt OR dipar.KPV5_ON.flt,
cmd_on    := alg.KPV15_nOpen, cmd_off  := NOT alg.KPV15_nOpen);
//--------------------------------------------------------------------------

//АОсс: Авар.-выс. Обороты СТ > 9300 об/мин
crs.Nst_HH(
in        := acpar.Nst.setpoint.HH,
brk       := FALSE,
cmd_on    := TRUE, cmd_off  := FALSE);
//--------------------------------------------------------------------------

//АОбс: Авар.-выс. Обороты ТК > 8400 об/мин
crs.Ntk_Av_HH(
in        := acpar.Ntk.setpoint.HH,
brk       := FALSE,
cmd_on    := TRUE, cmd_off  := FALSE);
//--------------------------------------------------------------------------

//АОбс: Отказ всех датчиков ЧВ ТК
crs.Ntk_flt(
in        := aipar.Ntk_1.flt AND aipar.Ntk_2.flt OR acpar.Ntk.flt,
brk       := FALSE,
cmd_on    := TRUE, cmd_off  := FALSE);
//--------------------------------------------------------------------------

//АОбс: Отказ всех датчиков ЧВ СТ
crs.Nst_flt(
in        := aipar.Nst_1.flt AND aipar.Nst_2.flt OR acpar.Nst.flt,
brk       := FALSE,
cmd_on    := TRUE, cmd_off  := FALSE);
//--------------------------------------------------------------------------

//АОбс: Авар.-выс. Температура газа на входе СТ
crs.Tg_inST_HH(
in        := acpar.Tg_inST.setpoint.HH,
brk       := FALSE,
cmd_on    := TRUE, cmd_off  := FALSE);
//--------------------------------------------------------------------------

//АОсс: Пожар ОД
crs.Fire_OD(
in        := dipar.Fire_OD.value,
brk       := dipar.Fire_OD.flt,
cmd_on    := TRUE, cmd_off  := FALSE);
//--------------------------------------------------------------------------

//АОбс: Авар.-выс. Высокая неравномерность 1-ой термопары
crs.Tg1_inSTdistort_HH(
in        := ABS ( acpar.Tg_inST.value - aipar.Tg_inST_1.value ) > 100.0,
brk       := aipar.Tg_inST_1.flt,
cmd_on    := am.SK.isON, cmd_off  := am.SK.isOFF);
//--------------------------------------------------------------------------

//АОбс: Авар.-выс. Высокая неравномерность 2-ой термопары
crs.Tg2_inSTdistort_HH(
in        := ABS ( acpar.Tg_inST.value - aipar.Tg_inST_2.value ) > 100.0,
brk       := aipar.Tg_inST_2.flt,
cmd_on    := am.SK.isON, cmd_off  := am.SK.isOFF);
//--------------------------------------------------------------------------

//АОбс: Авар.-выс. Высокая неравномерность 3-ой термопары
crs.Tg3_inSTdistort_HH(
in        := ABS ( acpar.Tg_inST.value - aipar.Tg_inST_3.value ) > 100.0,
brk       := aipar.Tg_inST_3.flt,
cmd_on    := am.SK.isON, cmd_off  := am.SK.isOFF);
//--------------------------------------------------------------------------

//АОбс: Авар.-выс. Высокая неравномерность 4-ой термопары
crs.Tg4_inSTdistort_HH(
in        := ABS ( acpar.Tg_inST.value - aipar.Tg_inST_4.value ) > 100.0,
brk       := aipar.Tg_inST_4.flt,
cmd_on    := am.SK.isON, cmd_off  := am.SK.isOFF);
//--------------------------------------------------------------------------

//АОбс: Авар.-выс. Высокая неравномерность 5-ой термопары
crs.Tg5_inSTdistort_HH(
in        := ABS ( acpar.Tg_inST.value - aipar.Tg_inST_5.value ) > 100.0,
brk       := aipar.Tg_inST_5.flt,
cmd_on    := am.SK.isON, cmd_off  := am.SK.isOFF);
//--------------------------------------------------------------------------

//АОбс: Авар.-выс. Высокая неравномерность 6-ой термопары
crs.Tg6_inSTdistort_HH(
in        := ABS ( acpar.Tg_inST.value - aipar.Tg_inST_6.value ) > 100.0,
brk       := aipar.Tg_inST_6.flt,
cmd_on    := am.SK.isON, cmd_off  := am.SK.isOFF);
//--------------------------------------------------------------------------

//АОбс: Отказ 4-х и более термопар
crs.Tg_inSTflt(
in        := alg.TstInWork < 3,
brk       := FALSE,
cmd_on    := TRUE, cmd_off  := FALSE);
//--------------------------------------------------------------------------

//АОбс: Нет розжига на пуске
crs.nIgnition(
in        := NOT FuelReg.fReg.isFire,
brk       := FALSE,
cmd_on    := alg.sh_nIgnition, cmd_off  := NOT alg.sh_nIgnition);
//--------------------------------------------------------------------------

//АОбс: Погасание факела
crs.Fire_flt(
in        := FuelReg.fReg.noFire,
brk       := FALSE,
cmd_on    := TRUE, cmd_off  := FALSE);
//--------------------------------------------------------------------------

//АОбс: Отсутствие раскрутки ТК
crs.Ntk_nBoost(
in        := acpar.Ntk.value < 5600,
brk       := acpar.Ntk.flt,
cmd_on    := alg.sh_nBoost, cmd_off  := NOT alg.sh_nBoost);
//--------------------------------------------------------------------------

//АОбс: Рассогласование ДГ
crs.DGdistort(
in        := ABS(aopar.DG_set.value - aipar.DG_Pos.value) >= 1.0,
brk       := aipar.DG_Pos.flt,
cmd_on    := am.SK.on, cmd_off  := NOT am.SK.on);
//--------------------------------------------------------------------------

//АОбс: Авар.-выс. Давление воздуха за 14-й ступенью осевого компрессора
crs.Pa_out14_HH(
in        := aipar.Pa_out14.setpoint.HH,
brk       := aipar.Pa_out14.flt,
cmd_on    := TRUE, cmd_off  := FALSE);
//--------------------------------------------------------------------------

//АОбс: Неисправность БЗА на пуске
crs.BZA_ready_2(
in        := NOT dipar.BZA_ready_1.value OR NOT dipar.BZA_ready_2.value,
brk       := FALSE,
cmd_on    := ( acpar.Ntk.value > BZA.Ntk_SetUp ) AND ( acpar.Nst.value > BZA.Nst_SetUp ), cmd_off  := NOT tch.GTDstart.value);
//--------------------------------------------------------------------------

//АОсс: БЗА: Авария
crs.BZA_alr(
in        := dipar.BZA_alr.value,
brk       := dipar.BZA_alr.flt,
cmd_on    := TRUE, cmd_off  := FALSE);
//--------------------------------------------------------------------------

//==========================================================================

//==========================================================================
//Подсистема: Маслосистема двигателя
//--------------------------------------------------------------------------
//АОбс: Давление масла смазки ТК аварийное
crs.Pm_TK_An(
in        := dipar.Pm_TK_An.value,
brk       := dipar.Pm_TK_An.flt,
cmd_on    := alg.sh_PmGTD, cmd_off  := NOT alg.sh_PmGTD);
//--------------------------------------------------------------------------

//АОбс: Давление масла смазки СТ аварийное
crs.Pm_ST_An(
in        := dipar.Pm_ST_An.value,
brk       := dipar.Pm_ST_An.flt,
cmd_on    := alg.sh_PmGTD, cmd_off  := NOT alg.sh_PmGTD);
//--------------------------------------------------------------------------

//АОбс: Авар.-выс. Температура масла на выходе двигателя
crs.Tm_outD_HH(
in        := aipar.Tm_outD.setpoint.HH,
brk       := aipar.Tm_outD.flt,
cmd_on    := TRUE, cmd_off  := FALSE);
//--------------------------------------------------------------------------

//АОсс: Стружка в масле на выходе Д
crs.Chip_outD(
in        := dipar.Chip_outD.value,
brk       := dipar.Chip_outD.flt,
cmd_on    := TRUE, cmd_off  := FALSE);
//--------------------------------------------------------------------------

//==========================================================================

//==========================================================================
//Подсистема: Воздушный стартер
//--------------------------------------------------------------------------
//АОбс: Аварийное давление газа до крана 13
crs.Pg_InKR13(
in        := dipar.Pg_InKR13.value,
brk       := dipar.Pg_InKR13.flt,
cmd_on    := alg.sh_Pg_InKR13, cmd_off  := NOT alg.sh_Pg_InKR13);
//--------------------------------------------------------------------------

//АОбс: Давление масла смазки воздушного стартера высокий уровень
crs.Pm_Starter_Av(
in        := dipar.Pm_Starter_Av.value,
brk       := dipar.Pm_Starter_Av.flt,
cmd_on    := TRUE, cmd_off  := FALSE);
//--------------------------------------------------------------------------

//АОбс: Давление масла смазки воздушного стартера низкий уровень
crs.Pm_Starter_An(
in        := dipar.Pm_Starter_An.value,
brk       := dipar.Pm_Starter_An.flt,
cmd_on    := alg.sh_Starter, cmd_off  := am.KR13.isOFF);
//--------------------------------------------------------------------------

//==========================================================================

//==========================================================================
//Подсистема: Аппарат воздушного охлаждения масла двигателя
//--------------------------------------------------------------------------
//==========================================================================

//==========================================================================
//Подсистема: Блок топливного газа
//--------------------------------------------------------------------------
//АОбс: Давление газа перед дозатором газа Аварийное
crs.Ptg_inDG_An(
in        := dipar.Ptg_inDG_An.value,
brk       := dipar.Ptg_inDG_An.flt,
cmd_on    := alg.sh_TG, cmd_off  := NOT alg.sh_TG);
//--------------------------------------------------------------------------

//АОсс: dP перед форсунками камеры сгорания >10кПа
crs.dP_F_Pv(
in        := dipar.dP_F_Pv.value,
brk       := dipar.dP_F_Pv.flt,
cmd_on    := am.SK.isOFF AND ( acpar.Ntk.value < 100 ), cmd_off  := am.SK.isON);
//--------------------------------------------------------------------------

//АОбс: Аварийное давление масла перед ДГ
crs.Pm_SAR_An(
in        := dipar.Pm_SAR_An.value,
brk       := dipar.Pm_SAR_An.flt,
cmd_on    := alg.sh_SAR, cmd_off  := NOT alg.sh_SAR);
//--------------------------------------------------------------------------

//АОбс: Авар.-низ. Давление топливного газа перед ТРК
crs.Ptg_inTRK_LL(
in        := aipar.Ptg_inTRK.setpoint.LL,
brk       := aipar.Ptg_inTRK.flt,
cmd_on    := alg.sh_TG, cmd_off  := NOT alg.sh_TG);
//--------------------------------------------------------------------------

//==========================================================================

//==========================================================================
//Подсистема: Блок пускового газа
//--------------------------------------------------------------------------
//==========================================================================

//==========================================================================
//Подсистема: Противообледенительная система и воздухоочистное устройство
//--------------------------------------------------------------------------
//==========================================================================

//==========================================================================
//Подсистема: Компрессорная установка/блок нагнетателя
//--------------------------------------------------------------------------
//АОсс: Помпаж нагнетателя
crs.AS_Av(
in        := s_tunpar.ASprot.surge,
brk       := s_tunpar.ASprot.surgeAlertBrk,
cmd_on    := TRUE, cmd_off  := FALSE);
//--------------------------------------------------------------------------

//АОсс: Авар.-низ. Перепад давления “масло-газ”
crs.dPmg_LL(
in        := aipar.dPmg.setpoint.LL OR dipar.dPmg_An.value,
brk       := dipar.dPmg_An.flt OR aipar.dPmg.flt OR NOT aipar.dPmg.setpoint.isLL,
cmd_on    := alg.sh_dPmg, cmd_off  := NOT alg.sh_dPmg);
//--------------------------------------------------------------------------

//АОсс: Давление масла смазки Н аварийное
crs.Pm_N_An(
in        := dipar.Pm_N_An.value,
brk       := dipar.Pm_N_An.flt,
cmd_on    := alg.sh_PmN, cmd_off  := NOT alg.sh_PmN);
//--------------------------------------------------------------------------

//АОсс: Аварийный осевой сдвиг ротора Н
crs.Zs_Nl(
in        := dipar.Zs_Nl.value,
brk       := dipar.Zs_Nl.flt,
cmd_on    := TRUE, cmd_off  := FALSE);
//--------------------------------------------------------------------------

//АОбс: Кран 6 закрыт на пуске
crs.Kr6_off_start(
in        := dipar.Kr6_off.value,
brk       := dipar.Kr6_off.flt,
cmd_on    := acpar.Nst.value > 300.0  AND Start_D.drm.active, cmd_off  := acpar.Nst.value < 300.0 OR NOT Start_D.drm.active);
//--------------------------------------------------------------------------

//==========================================================================

//==========================================================================
//Подсистема: Блок управления
//--------------------------------------------------------------------------
//==========================================================================

//==========================================================================
//Подсистема: Газовая обвязка
//--------------------------------------------------------------------------
//АОбс: Самопроизвольное закрытие крана 1
crs.Causeless_KR1_off(
in        := NOT dipar.Kr1_ON.value,
brk       := FALSE,
cmd_on    := alg.work, cmd_off  := NOT alg.work);
//--------------------------------------------------------------------------

//АОбс: Самопроизвольное закрытие крана 2
crs.Causeless_KR2_off(
in        := NOT dipar.Kr2_ON.value AND dipar.Kr6_off.value,
brk       := FALSE,
cmd_on    := alg.work, cmd_off  := NOT alg.work);
//--------------------------------------------------------------------------

//АОбс: Самопроизвольное закрытие крана 6
crs.Causeless_KR6_off(
in        := NOT dipar.Kr6_ON.value AND (NOT dipar.Kr2_ON.value OR dipar.Kr2_off.value),
brk       := FALSE,
cmd_on    := alg.work, cmd_off  := NOT alg.work);
//--------------------------------------------------------------------------

//АОбс: Самопроизвольная перестановка кранов 10, 11
crs.Causeless_KR10_11(
in        := NOT ( dipar.Kr10_off.value AND dipar.Kr11_ON.value ),
brk       := FALSE,
cmd_on    := am.KR15.on, cmd_off  := NOT am.KR15.on);
//--------------------------------------------------------------------------

//==========================================================================

//==========================================================================
//Подсистема: Контроль защит
//--------------------------------------------------------------------------

                  
END_FUNCTION

{region INFO}
(*
 Назначение: Используется для вызова предпусковых условий
 Автор:  /Andrey/ 24.06.2025 16:50:31
 Версия: v00.00.22
 Проект: KA107__GPA2
*)
{endregion}
FUNCTION ppu_update : BOOL
VAR_INPUT
END_VAR

                    //==========================================================================

//==========================================================================
//Подсистема: Внешние источники
//--------------------------------------------------------------------------
//Есть недеблокированные АС
ppu.crs_aggregated(
in     := crs.common.aggregated,
cmd_on := ppu.check_HR.value, cmd_off  := NOT ppu.check_HR.value);
//--------------------------------------------------------------------------

//==========================================================================

//==========================================================================
//Подсистема: Блок двигателя
//--------------------------------------------------------------------------
//Расчетная N ротора ГГ > 100 об/мин
ppu.evNvd_H(
in     := acpar.Ntk.value > 100.0,
cmd_on := ppu.check_HR.value, cmd_off  := NOT ppu.check_HR.value);
//--------------------------------------------------------------------------

//Расчетная N ротора СТ > 100 об/мин
ppu.evNst_H(
in     := acpar.Nst.value > 100.0,
cmd_on := ppu.check_HR.value, cmd_off  := NOT ppu.check_HR.value);
//--------------------------------------------------------------------------

//Нет сигнала: СК закрыт
ppu.N_SK_off(
in     := NOT dipar.SK_off.value,
cmd_on := ppu.check_HR.value, cmd_off  := NOT ppu.check_HR.value);
//--------------------------------------------------------------------------

//Загазованность контейнеров выше нормы
ppu.Zagaz_OD_Pv(
in     := dipar.Zagaz_OD_Pv.value,
cmd_on := ppu.check_HR.value, cmd_off  := NOT ppu.check_HR.value);
//--------------------------------------------------------------------------

//Сигнализатор обледенения
ppu.Ace_alr(
in     := dipar.Ace_alr.value,
cmd_on := ppu.check_GR.value, cmd_off  := NOT ppu.check_GR.value);
//--------------------------------------------------------------------------

//Нет сигнала: ТРК: готовность
ppu.N_TRKready(
in     := NOT dipar.TRKready.value,
cmd_on := ppu.check_HR.value, cmd_off  := NOT ppu.check_HR.value);
//--------------------------------------------------------------------------

//ТРК: авария
ppu.TRKalr(
in     := dipar.TRKalr.value,
cmd_on := ppu.check_HR.value, cmd_off  := NOT ppu.check_HR.value);
//--------------------------------------------------------------------------

//Нет сигнала: БЗА: Готовность 1
ppu.N_BZA_ready_1(
in     := NOT dipar.BZA_ready_1.value,
cmd_on := ppu.check_GR.value, cmd_off  := NOT ppu.check_GR.value);
//--------------------------------------------------------------------------

//Неисправность БЗА
ppu.BZA_flt(
in     := dipar.BZA_ready_1.value AND dipar.BZA_ready_2.value,
cmd_on := ppu.check_GR.value, cmd_off  := NOT ppu.check_GR.value);
//--------------------------------------------------------------------------

//==========================================================================

//==========================================================================
//Подсистема: Маслосистема двигателя
//--------------------------------------------------------------------------
//Пониж. Температура масла в баке Д и Н
ppu.Tm_MB_L(
in     := aipar.Tm_MB.setpoint.L,
cmd_on := ppu.check_HR.value, cmd_off  := NOT ppu.check_HR.value);
//--------------------------------------------------------------------------

//==========================================================================

//==========================================================================
//Подсистема: Воздушный стартер
//--------------------------------------------------------------------------
//==========================================================================

//==========================================================================
//Подсистема: Аппарат воздушного охлаждения масла двигателя
//--------------------------------------------------------------------------
//==========================================================================

//==========================================================================
//Подсистема: Блок топливного газа
//--------------------------------------------------------------------------
//Кран №9 не открыт
ppu.Kr9_ON(
in     := NOT dipar.Kr9_ON.value OR dipar.Kr9_off.value,
cmd_on := ppu.check_HR.value, cmd_off  := NOT ppu.check_HR.value);
//--------------------------------------------------------------------------

//Кран №12 не закрыт
ppu.Kr12_off(
in     := NOT dipar.Kr12_off.value OR dipar.Kr12_ON.value,
cmd_on := ppu.check_HR.value, cmd_off  := NOT ppu.check_HR.value);
//--------------------------------------------------------------------------

//==========================================================================

//==========================================================================
//Подсистема: Блок пускового газа
//--------------------------------------------------------------------------
//Кран №10 не открыт
ppu.Kr10_ON(
in     := NOT dipar.Kr10_ON.value OR dipar.Kr10_off.value,
cmd_on := ppu.check_HR.value, cmd_off  := NOT ppu.check_HR.value);
//--------------------------------------------------------------------------

//Кран №11 не закрыт
ppu.Kr11_off(
in     := NOT dipar.Kr11_off.value OR dipar.Kr11_ON.value,
cmd_on := ppu.check_HR.value, cmd_off  := NOT ppu.check_HR.value);
//--------------------------------------------------------------------------

//==========================================================================

//==========================================================================
//Подсистема: Противообледенительная система и воздухоочистное устройство
//--------------------------------------------------------------------------
//==========================================================================

//==========================================================================
//Подсистема: Компрессорная установка/блок нагнетателя
//--------------------------------------------------------------------------
//Пониж. Температура масла в баке уплотнения
ppu.Tm_MBU_L(
in     := aipar.Tm_MBU.setpoint.L,
cmd_on := ppu.check_HR.value, cmd_off  := NOT ppu.check_HR.value);
//--------------------------------------------------------------------------

//==========================================================================

//==========================================================================
//Подсистема: Блок управления
//--------------------------------------------------------------------------
//Нет сигнала: Предохранитель UCP1-XTFU1:1 питания модулей AO исправен
ppu.N_Fuse_AO_UCP1(
in     := NOT dipar.Fuse_AO_UCP1.value,
cmd_on := ppu.check_HR.value, cmd_off  := NOT ppu.check_HR.value);
//--------------------------------------------------------------------------

//Нет сигнала: Предохранитель UCP1-XTFU1:2 питания модулей DO исправен
ppu.N_Fuse_DO_UCP1(
in     := NOT dipar.Fuse_DO_UCP1.value,
cmd_on := ppu.check_HR.value, cmd_off  := NOT ppu.check_HR.value);
//--------------------------------------------------------------------------

//Нет сигнала: Предохранитель UCP1--XTFU6:1 питания датчиков температуры и влажности
ppu.N_Fuse_Air_UCP1(
in     := NOT dipar.Fuse_Air_UCP1.value,
cmd_on := ppu.check_HR.value, cmd_off  := NOT ppu.check_HR.value);
//--------------------------------------------------------------------------

//Нет сигнала: Предохранитель UE1-XTFU1:2 питания модулей DO исправен
ppu.N_Fuse_DO_UE1(
in     := NOT dipar.Fuse_DO_UE1.value,
cmd_on := ppu.check_HR.value, cmd_off  := NOT ppu.check_HR.value);
//--------------------------------------------------------------------------

//Перегрузка фильтра EV1 (Осн.)
ppu.EV1(
in     := dipar.EV1.value,
cmd_on := ppu.check_HR.value, cmd_off  := NOT ppu.check_HR.value);
//--------------------------------------------------------------------------

//Перегрузка фильтра EV2 (Рез.)
ppu.EV2(
in     := dipar.EV2.value,
cmd_on := ppu.check_HR.value, cmd_off  := NOT ppu.check_HR.value);
//--------------------------------------------------------------------------

//Нет сигнала: Контроль основного ввода питания (-KV1)
ppu.N_U_main(
in     := NOT dipar.U_main.value,
cmd_on := ppu.check_HR.value, cmd_off  := NOT ppu.check_HR.value);
//--------------------------------------------------------------------------

//Нет сигнала: Контроль резервного ввода питания (-KV2)
ppu.N_U_res(
in     := NOT dipar.U_res.value,
cmd_on := ppu.check_HR.value, cmd_off  := NOT ppu.check_HR.value);
//--------------------------------------------------------------------------

//Нет сигнала: Контроль -AG1
ppu.N_AG1(
in     := NOT dipar.AG1.value,
cmd_on := ppu.check_HR.value, cmd_off  := NOT ppu.check_HR.value);
//--------------------------------------------------------------------------

//Нет сигнала: Контроль -AG2
ppu.N_AG2(
in     := NOT dipar.AG2.value,
cmd_on := ppu.check_HR.value, cmd_off  := NOT ppu.check_HR.value);
//--------------------------------------------------------------------------

//Нет сигнала: Контроль -AG3
ppu.N_AG3(
in     := NOT dipar.AG3.value,
cmd_on := ppu.check_HR.value, cmd_off  := NOT ppu.check_HR.value);
//--------------------------------------------------------------------------

//Нет сигнала: Контроль -AG4
ppu.N_AG4(
in     := NOT dipar.AG4.value,
cmd_on := ppu.check_HR.value, cmd_off  := NOT ppu.check_HR.value);
//--------------------------------------------------------------------------

//Нет сигнала: Контроль -AG9
ppu.N_AG9(
in     := NOT dipar.AG9.value,
cmd_on := ppu.check_HR.value, cmd_off  := NOT ppu.check_HR.value);
//--------------------------------------------------------------------------

//Нет сигнала: Контроль -AG10
ppu.N_AG10(
in     := NOT dipar.AG10.value,
cmd_on := ppu.check_HR.value, cmd_off  := NOT ppu.check_HR.value);
//--------------------------------------------------------------------------

//Нет сигнала: Контроль -AG15
ppu.N_AG15(
in     := NOT dipar.AG15.value,
cmd_on := ppu.check_HR.value, cmd_off  := NOT ppu.check_HR.value);
//--------------------------------------------------------------------------

//Нет сигнала: Контроль -AG16
ppu.N_AG16(
in     := NOT dipar.AG16.value,
cmd_on := ppu.check_HR.value, cmd_off  := NOT ppu.check_HR.value);
//--------------------------------------------------------------------------

//Нет сигнала: Контроль -AG5
ppu.N_AG5(
in     := NOT dipar.AG5.value,
cmd_on := ppu.check_HR.value, cmd_off  := NOT ppu.check_HR.value);
//--------------------------------------------------------------------------

//Нет сигнала: Контроль -AG6
ppu.N_AG6(
in     := NOT dipar.AG6.value,
cmd_on := ppu.check_HR.value, cmd_off  := NOT ppu.check_HR.value);
//--------------------------------------------------------------------------

//Нет сигнала: Контроль -AG8
ppu.N_AG8(
in     := NOT dipar.AG8.value,
cmd_on := ppu.check_HR.value, cmd_off  := NOT ppu.check_HR.value);
//--------------------------------------------------------------------------

//Нет сигнала: Контроль -AG17
ppu.N_AG17(
in     := NOT dipar.AG17.value,
cmd_on := ppu.check_HR.value, cmd_off  := NOT ppu.check_HR.value);
//--------------------------------------------------------------------------

//Нет сигнала: Контроль -AG18
ppu.N_AG18(
in     := NOT dipar.AG18.value,
cmd_on := ppu.check_HR.value, cmd_off  := NOT ppu.check_HR.value);
//--------------------------------------------------------------------------

//Нет сигнала: Контроль питания ПРУ
ppu.N_U_PRU(
in     := NOT dipar.U_PRU.value,
cmd_on := ppu.check_HR.value, cmd_off  := NOT ppu.check_HR.value);
//--------------------------------------------------------------------------

//Нет сигнала: Контроль питания ТРК осн.
ppu.N_Utrk_main(
in     := NOT dipar.Utrk_main.value,
cmd_on := ppu.check_HR.value, cmd_off  := NOT ppu.check_HR.value);
//--------------------------------------------------------------------------

//Контроль замыкания на землю питания ИМ
ppu.U_G_AM(
in     := dipar.U_G_AM.value,
cmd_on := ppu.check_HR.value, cmd_off  := NOT ppu.check_HR.value);
//--------------------------------------------------------------------------

//Нет сигнала: Контроль питания AI
ppu.N_U_AI(
in     := NOT dipar.U_AI.value,
cmd_on := ppu.check_HR.value, cmd_off  := NOT ppu.check_HR.value);
//--------------------------------------------------------------------------

//Нет сигнала: Контроль питания DI
ppu.N_U_DI(
in     := NOT dipar.U_DI.value,
cmd_on := ppu.check_HR.value, cmd_off  := NOT ppu.check_HR.value);
//--------------------------------------------------------------------------

//Нет сигнала: Контроль питания БИЗ
ppu.N_U_BIZ(
in     := NOT dipar.U_BIZ.value,
cmd_on := ppu.check_HR.value, cmd_off  := NOT ppu.check_HR.value);
//--------------------------------------------------------------------------

//Нет сигнала: Контроль питания ИМ
ppu.N_U_AM(
in     := NOT dipar.U_AM.value,
cmd_on := ppu.check_HR.value, cmd_off  := NOT ppu.check_HR.value);
//--------------------------------------------------------------------------

//Нет сигнала: Контроль питания аппаратуры вибрации, =24 В
ppu.N_Uvs_24(
in     := NOT dipar.Uvs_24.value,
cmd_on := ppu.check_HR.value, cmd_off  := NOT ppu.check_HR.value);
//--------------------------------------------------------------------------

//Нет сигнала: Контроль питания дополнительного оборудования, =24В
ppu.N_Uother_24(
in     := NOT dipar.Uother_24.value,
cmd_on := ppu.check_HR.value, cmd_off  := NOT ppu.check_HR.value);
//--------------------------------------------------------------------------

//Нет сигнала: Контроль питания ИМ2
ppu.N_U_AM2(
in     := NOT dipar.U_AM2.value,
cmd_on := ppu.check_HR.value, cmd_off  := NOT ppu.check_HR.value);
//--------------------------------------------------------------------------

//Нет сигнала: Контроль питания ТРК рез.
ppu.N_Utrk_res(
in     := NOT dipar.Utrk_res.value,
cmd_on := ppu.check_HR.value, cmd_off  := NOT ppu.check_HR.value);
//--------------------------------------------------------------------------

//БЭО. Перегрузка фильтра EV3 (Осн. БЭО)
ppu.EV3(
in     := dipar.EV3.value,
cmd_on := ppu.check_HR.value, cmd_off  := NOT ppu.check_HR.value);
//--------------------------------------------------------------------------

//БЭО. Перегрузка фильтра EV4 (Рез. БЭО)
ppu.EV4(
in     := dipar.EV4.value,
cmd_on := ppu.check_HR.value, cmd_off  := NOT ppu.check_HR.value);
//--------------------------------------------------------------------------

//Нет сигнала: БЭО. Контроль основного ввода питания БЭО (-KV3)
ppu.N_Ubeo_main(
in     := NOT dipar.Ubeo_main.value,
cmd_on := ppu.check_HR.value, cmd_off  := NOT ppu.check_HR.value);
//--------------------------------------------------------------------------

//Нет сигнала: БЭО. Контроль резервного ввода питания БЭО (-KV4)
ppu.N_Ubeo_res(
in     := NOT dipar.Ubeo_res.value,
cmd_on := ppu.check_HR.value, cmd_off  := NOT ppu.check_HR.value);
//--------------------------------------------------------------------------

//Нет сигнала: БЭО. Контроль -AG11
ppu.N_AG11(
in     := NOT dipar.AG11.value,
cmd_on := ppu.check_HR.value, cmd_off  := NOT ppu.check_HR.value);
//--------------------------------------------------------------------------

//Нет сигнала: БЭО. Контроль -AG12
ppu.N_AG12(
in     := NOT dipar.AG12.value,
cmd_on := ppu.check_HR.value, cmd_off  := NOT ppu.check_HR.value);
//--------------------------------------------------------------------------

//БЭО. Контроль замыкания на землю питания БЭО (-KR5)
ppu.U_G_KR5(
in     := dipar.U_G_KR5.value,
cmd_on := ppu.check_HR.value, cmd_off  := NOT ppu.check_HR.value);
//--------------------------------------------------------------------------

//Нет сигнала: БЭО. Контроль питания кн. ЭАО
ppu.N_U_KEAO(
in     := NOT dipar.U_KEAO.value,
cmd_on := ppu.check_HR.value, cmd_off  := NOT ppu.check_HR.value);
//--------------------------------------------------------------------------

//Нет сигнала: БЭО. Контроль питания БЭО
ppu.N_U_BEO(
in     := NOT dipar.U_BEO.value,
cmd_on := ppu.check_HR.value, cmd_off  := NOT ppu.check_HR.value);
//--------------------------------------------------------------------------

//Нет сигнала: БЭО. Контроль питания БЗА
ppu.N_U_BZA(
in     := NOT dipar.U_BZA.value,
cmd_on := ppu.check_HR.value, cmd_off  := NOT ppu.check_HR.value);
//--------------------------------------------------------------------------

//Ошибка -AUO1
ppu.Err_AUO1(
in     := dipar.Err_AUO1.value,
cmd_on := ppu.check_HR.value, cmd_off  := NOT ppu.check_HR.value);
//--------------------------------------------------------------------------

//==========================================================================

//==========================================================================
//Подсистема: Газовая обвязка
//--------------------------------------------------------------------------
//Кран №1 не закрыт
ppu.Kr1_off(
in     := NOT dipar.Kr1_off.value OR dipar.Kr1_ON.value,
cmd_on := ppu.check_HR.value, cmd_off  := NOT ppu.check_HR.value);
//--------------------------------------------------------------------------

//Кран №2 не закрыт
ppu.Kr2_off(
in     := NOT dipar.Kr2_off.value OR dipar.Kr2_ON.value,
cmd_on := ppu.check_HR.value, cmd_off  := NOT ppu.check_HR.value);
//--------------------------------------------------------------------------

//Кран №4 не закрыт
ppu.Kr4_off(
in     := (NOT dipar.Kr4_off.value OR dipar.Kr4_ON.value) AND tch.nGas_N.value,
cmd_on := ppu.check_HR.value, cmd_off  := NOT ppu.check_HR.value);
//--------------------------------------------------------------------------

//Кран №5 не открыт
ppu.Kr5_ON(
in     := (NOT dipar.Kr5_ON.value OR dipar.Kr5_off.value) AND tch.nGas_N.value,
cmd_on := ppu.check_HR.value, cmd_off  := NOT ppu.check_HR.value);
//--------------------------------------------------------------------------

//Кран №5 не закрыт
ppu.Kr5_off(
in     := (NOT dipar.Kr5_off.value OR dipar.Kr5_ON.value) AND tch.Gas_N.value,
cmd_on := ppu.check_HR.value, cmd_off  := NOT ppu.check_HR.value);
//--------------------------------------------------------------------------

//Кран №6 не закрыт
ppu.Kr6_off(
in     := (NOT dipar.Kr6_off.value OR dipar.Kr6_ON.value) AND tch.nGas_N.value,
cmd_on := ppu.check_HR.value, cmd_off  := NOT ppu.check_HR.value);
//--------------------------------------------------------------------------

//==========================================================================

//==========================================================================
//Подсистема: Контроль защит
//--------------------------------------------------------------------------

                  
END_FUNCTION

{region INFO}
(*
 Назначение:   Используется для обработки аналоговых ИМов
 Автор:        /Разработчик/ 08.08.2025 8:32:24
 Конфигуратор: v00.01.00
 Проект:       KA107
*)
{endregion}
FUNCTION ama_update : BOOL
VAR_INPUT
END_VAR
VAR
END_VAR

                    //Дозатор газа
//Тип: a
am.DG.DU_prm := alg.V_000;
//У ИМа не генерируется вызов ФБ: am.DG();
//--------------------------------------------------------------------------

                  
END_FUNCTION

{region INFO}
(*
 Назначение:   Используется для обработки дискретных ИМов
 Автор:        /Разработчик/ 08.08.2025 8:32:24
 Конфигуратор: v00.01.00
 Проект:       KA107
*)
{endregion}
FUNCTION am_update : BOOL
VAR_INPUT
END_VAR
VAR
END_VAR

                    //Вытяжной вентилятор ВОУ
//Тип: 2x1
am.VV_VOU(
	DU_prm := true,
	onSigFlt := dipar.VV_VOU_on.flt,
	onSig := dipar.VV_VOU_on.value,
	onSig_sim_on := dipar.VV_VOU_on.sim_on,
	onSig_sim_value := dipar.VV_VOU_on.sim_value,
	onFlt := dopar.VV_VOU_on.flt,
	offFlt := dopar.VV_VOU_off.flt);
dopar.VV_VOU_on.value := am.VV_VOU.onOUT;
dopar.VV_VOU_off.value := am.VV_VOU.offOUT;

//Вентилятор 1 АВОМ
//Тип: 2x1
am.Vn1_AVOM(
	DU_prm := true,
	onSigFlt := dipar.Vn1_AVOM_on.flt,
	onSig := dipar.Vn1_AVOM_on.value,
	onSig_sim_on := dipar.Vn1_AVOM_on.sim_on,
	onSig_sim_value := dipar.Vn1_AVOM_on.sim_value,
	onFlt := dopar.Vn1_AVOM_on.flt,
	offFlt := dopar.Vn1_AVOM_off.flt);
dopar.Vn1_AVOM_on.value := am.Vn1_AVOM.onOUT;
dopar.Vn1_AVOM_off.value := am.Vn1_AVOM.offOUT;

//Вентилятор 2 АВОМ
//Тип: 2x1
am.Vn2_AVOM(
	DU_prm := true,
	onSigFlt := dipar.Vn2_AVOM_on.flt,
	onSig := dipar.Vn2_AVOM_on.value,
	onSig_sim_on := dipar.Vn2_AVOM_on.sim_on,
	onSig_sim_value := dipar.Vn2_AVOM_on.sim_value,
	onFlt := dopar.Vn2_AVOM_on.flt,
	offFlt := dopar.Vn2_AVOM_off.flt);
dopar.Vn2_AVOM_on.value := am.Vn2_AVOM.onOUT;
dopar.Vn2_AVOM_off.value := am.Vn2_AVOM.offOUT;

//Вентилятор 3 АВОМ
//Тип: 2x1
am.Vn3_AVOM(
	DU_prm := true,
	onSigFlt := dipar.Vn3_AVOM_on.flt,
	onSig := dipar.Vn3_AVOM_on.value,
	onSig_sim_on := dipar.Vn3_AVOM_on.sim_on,
	onSig_sim_value := dipar.Vn3_AVOM_on.sim_value,
	onFlt := dopar.Vn3_AVOM_on.flt,
	offFlt := dopar.Vn3_AVOM_off.flt);
dopar.Vn3_AVOM_on.value := am.Vn3_AVOM.onOUT;
dopar.Vn3_AVOM_off.value := am.Vn3_AVOM.offOUT;

//Вентилятор 4 АВОМ
//Тип: 2x1
am.Vn4_AVOM(
	DU_prm := true,
	onSigFlt := dipar.Vn4_AVOM_on.flt,
	onSig := dipar.Vn4_AVOM_on.value,
	onSig_sim_on := dipar.Vn4_AVOM_on.sim_on,
	onSig_sim_value := dipar.Vn4_AVOM_on.sim_value,
	onFlt := dopar.Vn4_AVOM_on.flt,
	offFlt := dopar.Vn4_AVOM_off.flt);
dopar.Vn4_AVOM_on.value := am.Vn4_AVOM.onOUT;
dopar.Vn4_AVOM_off.value := am.Vn4_AVOM.offOUT;

//Кран 1
//Тип: 2x2
am.Kr1(
	DU_prm := alg.V_000,
	onSigFlt := dipar.Kr1_on.flt,
	onSig := dipar.Kr1_on.value,
	onSig_sim_on := dipar.Kr1_on.sim_on,
	onSig_sim_value := dipar.Kr1_on.sim_value,
	offSigFlt := dipar.Kr1_off.flt,
	offSig := dipar.Kr1_off.value,
	offSig_sim_on := dipar.Kr1_off.sim_on,
	offSig_sim_value := dipar.Kr1_off.sim_value,
	onFlt := dopar.Kr1_on.flt,
	offFlt := dopar.Kr1_off.flt);
dopar.Kr1_on.value := am.Kr1.onOUT;
dopar.Kr1_off.value := am.Kr1.offOUT;

//Кран 2
//Тип: 2x2
am.Kr2(
	DU_prm := alg.V_000,
	onSigFlt := dipar.Kr2_on.flt,
	onSig := dipar.Kr2_on.value,
	onSig_sim_on := dipar.Kr2_on.sim_on,
	onSig_sim_value := dipar.Kr2_on.sim_value,
	offSigFlt := dipar.Kr2_off.flt,
	offSig := dipar.Kr2_off.value,
	offSig_sim_on := dipar.Kr2_off.sim_on,
	offSig_sim_value := dipar.Kr2_off.sim_value,
	onFlt := dopar.Kr2_on.flt,
	offFlt := dopar.Kr2_off.flt);
dopar.Kr2_on.value := am.Kr2.onOUT;
dopar.Kr2_off.value := am.Kr2.offOUT;

//Кран 4
//Тип: 2x2
am.Kr4(
	DU_prm := alg.V_000,
	onSigFlt := dipar.Kr4_on.flt,
	onSig := dipar.Kr4_on.value,
	onSig_sim_on := dipar.Kr4_on.sim_on,
	onSig_sim_value := dipar.Kr4_on.sim_value,
	offSigFlt := dipar.Kr4_off.flt,
	offSig := dipar.Kr4_off.value,
	offSig_sim_on := dipar.Kr4_off.sim_on,
	offSig_sim_value := dipar.Kr4_off.sim_value,
	onFlt := dopar.Kr4_on.flt,
	offFlt := dopar.Kr4_off.flt);
dopar.Kr4_on.value := am.Kr4.onOUT;
dopar.Kr4_off.value := am.Kr4.offOUT;

//Кран 5
//Тип: 2x2
am.Kr5(
	DU_prm := alg.V_000,
	onSigFlt := dipar.Kr5_on.flt,
	onSig := dipar.Kr5_on.value,
	onSig_sim_on := dipar.Kr5_on.sim_on,
	onSig_sim_value := dipar.Kr5_on.sim_value,
	offSigFlt := dipar.Kr5_off.flt,
	offSig := dipar.Kr5_off.value,
	offSig_sim_on := dipar.Kr5_off.sim_on,
	offSig_sim_value := dipar.Kr5_off.sim_value,
	onFlt := dopar.Kr5_on.flt,
	offFlt := dopar.Kr5_off.flt);
dopar.Kr5_on.value := am.Kr5.onOUT;
dopar.Kr5_off.value := am.Kr5.offOUT;

//Кран 6
//Тип: 2x2
am.Kr6(
	DU_prm := alg.V_000 OR mde.M AND NOT dipar.Kr6_Off.value AND dipar.Kr2_ON.value,
	onSigFlt := dipar.Kr6_on.flt,
	onSig := dipar.Kr6_on.value,
	onSig_sim_on := dipar.Kr6_on.sim_on,
	onSig_sim_value := dipar.Kr6_on.sim_value,
	offSigFlt := dipar.Kr6_off.flt,
	offSig := dipar.Kr6_off.value,
	offSig_sim_on := dipar.Kr6_off.sim_on,
	offSig_sim_value := dipar.Kr6_off.sim_value,
	onFlt := dopar.Kr6_on.flt,
	offFlt := dopar.Kr6_off.flt);
dopar.Kr6_on.value := am.Kr6.onOUT;
dopar.Kr6_off.value := am.Kr6.offOUT;

//Кран 12
//Тип: 2x2
am.Kr12(
	DU_prm := alg.V_000,
	onSigFlt := dipar.Kr12_on.flt,
	onSig := dipar.Kr12_on.value,
	onSig_sim_on := dipar.Kr12_on.sim_on,
	onSig_sim_value := dipar.Kr12_on.sim_value,
	offSigFlt := dipar.Kr12_off.flt,
	offSig := dipar.Kr12_off.value,
	offSig_sim_on := dipar.Kr12_off.sim_on,
	offSig_sim_value := dipar.Kr12_off.sim_value,
	onFlt := dopar.Kr12_on.flt,
	offFlt := dopar.Kr12_off.flt);
dopar.Kr12_on.value := am.Kr12.onOUT;
dopar.Kr12_off.value := am.Kr12.offOUT;

//Кран 9
//Тип: 2x2
am.Kr9.DU_prm := FALSE;
//У ИМа не генерируется вызов ФБ: am.Kr9();

//Кран 11
//Тип: 2x2
am.Kr11(
	DU_prm := alg.V_000,
	onSigFlt := dipar.Kr11_on.flt,
	onSig := dipar.Kr11_on.value,
	onSig_sim_on := dipar.Kr11_on.sim_on,
	onSig_sim_value := dipar.Kr11_on.sim_value,
	offSigFlt := dipar.Kr11_off.flt,
	offSig := dipar.Kr11_off.value,
	offSig_sim_on := dipar.Kr11_off.sim_on,
	offSig_sim_value := dipar.Kr11_off.sim_value,
	onFlt := dopar.Kr11_on.flt,
	offFlt := dopar.Kr11_off.flt);
dopar.Kr11_on.value := am.Kr11.onOUT;
dopar.Kr11_off.value := am.Kr11.offOUT;

//Кран 10
//Тип: 2x2
am.Kr10.DU_prm := FALSE;
//У ИМа не генерируется вызов ФБ: am.Kr10();

//КПВ 1
//Тип: 1x2
am.KPV1.DU_prm := alg.V_000;
//У ИМа не генерируется вызов ФБ: am.KPV1();

//КПВ 2
//Тип: 1x2
am.KPV2.DU_prm := alg.V_000;
//У ИМа не генерируется вызов ФБ: am.KPV2();

//КПВ 3
//Тип: 1x2
am.KPV3.DU_prm := alg.V_000;
//У ИМа не генерируется вызов ФБ: am.KPV3();

//КПВ 4
//Тип: 1x2
am.KPV4(
	DU_prm := alg.V_000,
	onSigFlt := dipar.KPV4_on.flt,
	onSig := dipar.KPV4_on.value,
	onSig_sim_on := dipar.KPV4_on.sim_on,
	onSig_sim_value := dipar.KPV4_on.sim_value,
	offSigFlt := dipar.KPV4_off.flt,
	offSig := dipar.KPV4_off.value,
	offSig_sim_on := dipar.KPV4_off.sim_on,
	offSig_sim_value := dipar.KPV4_off.sim_value,
	onFlt := dopar.KPV4_off.flt);
dopar.KPV4_off.value := NOT am.KPV4.onOUT;
//--------------------------------------------------------------------------

//КПВ 5
//Тип: 1x2
am.KPV5.DU_prm := alg.V_000;
//У ИМа не генерируется вызов ФБ: am.KPV5();

//Стопорный клапан
//Тип: 1x2
am.SK.DU_prm := alg.V_000;
//У ИМа не генерируется вызов ФБ: am.SK();

//Пусковой насос смазки
//Тип: 2x1
am.PNS(
	DU_prm := true,
	onSigFlt := dipar.PNS_on.flt,
	onSig := dipar.PNS_on.value,
	onSig_sim_on := dipar.PNS_on.sim_on,
	onSig_sim_value := dipar.PNS_on.sim_value,
	onFlt := dopar.PNS_on.flt,
	offFlt := dopar.PNS_off.flt);
dopar.PNS_on.value := am.PNS.onOUT;
dopar.PNS_off.value := am.PNS.offOUT;

//Пусковой насос уплотнения
//Тип: 2x1
am.PNU(
	DU_prm := true,
	onSigFlt := dipar.PNU_on.flt,
	onSig := dipar.PNU_on.value,
	onSig_sim_on := dipar.PNU_on.sim_on,
	onSig_sim_value := dipar.PNU_on.sim_value,
	onFlt := dopar.PNU_on.flt,
	offFlt := dopar.PNU_off.flt);
dopar.PNU_on.value := am.PNU.onOUT;
dopar.PNU_off.value := am.PNU.offOUT;

//ВНА
//Тип: 1x0
am.VNA(
	DU_prm := alg.V_000,
	onFlt := dopar.VNA_on.flt);
dopar.VNA_on.value := am.VNA.onOUT;
//--------------------------------------------------------------------------

//Звуковая сигнализация
//Тип: 1x0
am.Sound(
	DU_prm := alg.V_000,
	onFlt := dopar.Sound_on.flt);
dopar.Sound_on.value := am.Sound.onOUT;
//--------------------------------------------------------------------------

//Агрегат зажигания
//Тип: 1x0
am.AZ(
	DU_prm := alg.V_000,
	onFlt := dopar.AZ_on.flt);
dopar.AZ_on.value := am.AZ.onOUT;
//--------------------------------------------------------------------------

//Обогрев ВНА
//Тип: 1x0
am.VNA_heat(
	DU_prm := alg.V_000,
	onFlt := dopar.VNA_heat_on.flt);
dopar.VNA_heat_on.value := am.VNA_heat.onOUT;
//--------------------------------------------------------------------------

//Кран 13
//Тип: 1x1
am.Kr13(
	DU_prm := alg.V_000,
	onSigFlt := dipar.Kr13_on.flt,
	onSig := dipar.Kr13_on.value,
	onSig_sim_on := dipar.Kr13_on.sim_on,
	onSig_sim_value := dipar.Kr13_on.sim_value,
	onFlt := dopar.Kr13_on.flt);
dopar.Kr13_on.value := am.Kr13.onOUT;
//--------------------------------------------------------------------------

//Кран 15
//Тип: 1x0
am.Kr15(
	DU_prm := alg.V_000,
	onFlt := dopar.Kr15_on.flt);
dopar.Kr15_on.value := am.Kr15.onOUT;
//--------------------------------------------------------------------------

//Вытяжной вентилятор нагнетателя
//Тип: 2x1
am.VVN(
	DU_prm := true,
	onSigFlt := dipar.VVN_on.flt,
	onSig := dipar.VVN_on.value,
	onSig_sim_on := dipar.VVN_on.sim_on,
	onSig_sim_value := dipar.VVN_on.sim_value,
	onFlt := dopar.VVN_on.flt,
	offFlt := dopar.VVN_off.flt);
dopar.VVN_on.value := am.VVN.onOUT;
dopar.VVN_off.value := am.VVN.offOUT;

                  
END_FUNCTION

{region INFO}
(*
 Назначение:   Используется для обработки расчетных аналоговых параметров
 Автор:        /Разработчик/ 08.08.2025 8:32:24
 Конфигуратор: v00.01.00
 Проект:       KA107
*)
{endregion}
FUNCTION acpar_update : BOOL
VAR_INPUT
END_VAR
VAR
END_VAR

                    acpar.Ntk(); //Расчётная Nтк
acpar.Nst(); //Расчётная Nст
acpar.Tg_inST(); //Расчётная Тг перед СТ
acpar.NtkPrived(); //Приведенная Nгг
acpar.Qtg_m3(); //Расход топливного газа

                  
END_FUNCTION

{region INFO}
(*
 Назначение:   Используется для обработки кнопок
 Автор:        /Разработчик/ 08.08.2025 8:32:24
 Конфигуратор: v00.01.00
 Проект:       KA107
*)
{endregion}
FUNCTION btn_update : BOOL
VAR_INPUT
END_VAR
VAR
END_VAR

                    //Имитацию включить
btn.imit_ON.prm := mde.Repair;
btn.imit_ON();

//Имитацию выключить
btn.imit_OF.prm := TRUE;
btn.imit_OF();

//Тестирование включить
btn.test_on.prm := mde.Repair;
btn.test_on();

//Тестирование выключить
btn.test_off.prm := TRUE;
btn.test_off();

//Ремонт
btn.Repair.prm := alg.V_000 AND NOT tch.PrepareStart.value;
btn.Repair();

//Холодный резерв
btn.HR.prm := ( mde.Repair OR mde.GR ) AND NOT tch.PrepareStart.value AND NOT tch.CheckAlarm_on.Value ;
btn.HR();

//Горячий резерв
btn.GR.prm := mde.Repair OR mde.HR AND NOT tch.CheckAlarm_on.Value ;
btn.GR();

//Комплексная проверка кранов
btn.KPK.prm := mde.GR AND NOT ( tch.PrepareStart.value OR tch.Gas_N.value );
btn.KPK();

//Холодная прокрутка
btn.HP.prm := mde.GR AND NOT tch.PrepareStart.value;
btn.HP();

//Автоматический пуск на Кольцо
btn.APK.prm := mde.GR AND NOT tch.PrepareStart.value;
btn.APK();

//Пуск
btn.Start.prm := check.ReadytoSF AND check.prm_start;
btn.Start();

//Отмена
btn.Cancel.prm := check.ReadytoSF OR mde.Repair OR check.tmrCancelPrm.Q;
btn.Cancel();

//Контроль САУ
btn.Check_SAU.prm := TRUE;
btn.Check_SAU();

//Переход Магистраль-Кольцо
btn.M_K.prm := mde.M OR mde.K_M;
btn.M_K();

//Переход Кольцо-Магистраль
btn.K_M.prm := mde.K OR mde.M_K;
btn.K_M();

//Нормальный останов со стравливанием
btn.NOss.prm := alg.work OR mde.NObs;
btn.NOss();

//Нормальный останов без стравливания
btn.NObs.prm := alg.work;
btn.NObs();

//Аварийный останов со стравливанием
btn.AOss.prm := TRUE;
btn.AOss();

//Аварийный останов без стравливания
btn.AObs.prm := NOT mde.AOss;
btn.AObs();

//Деблокировка
btn.Unlock.prm := TRUE;
btn.Unlock();

//РЧВ: вверх
btn.turnUP.prm := tch.GTDwork.value;
btn.turnUP();

//РЧВ: вниз
btn.turnDN.prm := tch.GTDwork.value;
btn.turnDN();

//Запись настроек регулятора
btn.set_tun.prm := NOT btn.get_tun.out;
btn.set_tun();

//Считывание настроек регулятора
btn.get_tun.prm := NOT btn.set_tun.out;
btn.get_tun();

//Стравливание
btn.bleeding.prm := alg.V_000;
btn.bleeding();

//Проверку защит включить
btn.CheckAlarm_on.prm := mde.Repair;
btn.CheckAlarm_on();

//Проверку защит выключить
btn.CheckAlarm_off.prm := mde.Repair;
btn.CheckAlarm_off();

                  
END_FUNCTION

{region INFO}
(*
 Назначение:   Используется для обработки режимов
 Автор:        /Разработчик/ 08.08.2025 8:32:24
 Конфигуратор: v00.01.00
 Проект:       KA107
*)
{endregion}
FUNCTION mde_update : BOOL
VAR_INPUT
END_VAR
VAR
END_VAR

                    alg.AOss_tech := FALSE;
alg.AObs_tech := FALSE;
alg.VOss_tech := FALSE;

IF
	   (mde.AObs) AND (alg.AOss) //Переход: АОбс->АОсс
	OR (mde.NOss) AND (alg.AOss OR alg.AObs) //Переход: НОсс->АОсс
	OR (mde.NObs) AND (alg.AOss) //Переход: НОбс->АОсс
	OR (mde.Repair) AND (alg.AOss AND tch.Gas_N.value) //Переход: Ремонт->АОсс
	OR (mde.HR) AND (alg.AOss AND tch.Gas_N.value) //Переход: ХР->АОсс
	OR (mde.GR) AND (alg.AOss AND tch.Gas_N.value) //Переход: ГР->АОсс
	OR (mde.AObs) AND (alg.AOss OR alg.AObs AND tch.nGas_N.value) //Переход: АОбс->АОсс
	OR (mde.PZ) AND (alg.AOss OR alg.AObs AND tch.nGas_N.value) //Переход: ПЗ->АОсс
	OR (mde.HP) AND (alg.AOss OR alg.AObs AND tch.nGas_N.value) //Переход: ХП->АОсс
	OR (mde.KPK) AND (alg.AOss OR alg.AObs AND tch.nGas_N.value) //Переход: КПК->АОсс
	OR (mde.APK) AND (alg.AOss OR alg.AObs AND tch.nGas_N.value) //Переход: АПК->АОсс
	OR (mde.K) AND (alg.AOss) //Переход: Кольцо->АОсс
	OR (mde.M) AND (alg.AOss) //Переход: Магистраль->АОсс
	OR (mde.K_M) AND (alg.AOss) //Переход: Переход К-М->АОсс
	OR (mde.M_K) AND (alg.AOss) //Переход: Переход М-К->АОсс
					THEN mde.number := enum_mode.AOss;

		IF
		   (mde.NOss) AND (alg.AObs)
		OR (mde.AObs) AND (alg.AObs AND tch.nGas_N.value)
		OR (mde.PZ) AND (alg.AObs AND tch.nGas_N.value)
		OR (mde.HP) AND (alg.AObs AND tch.nGas_N.value)
		OR (mde.KPK) AND (alg.AObs AND tch.nGas_N.value)
		OR (mde.APK) AND (alg.AObs AND tch.nGas_N.value)
					THEN alg.AOss_tech := TRUE;
		END_IF;
ELSIF
	   (mde.NObs) AND (alg.AObs) //Переход: НОбс->АОбс
	OR (mde.HP) AND (alg.AObs) //Переход: ХП->АОбс
	OR (mde.KPK) AND (alg.AObs) //Переход: КПК->АОбс
	OR (mde.APK) AND (alg.AObs) //Переход: АПК->АОбс
	OR (mde.K) AND (alg.AObs) //Переход: Кольцо->АОбс
	OR (mde.M) AND (alg.AObs) //Переход: Магистраль->АОбс
	OR (mde.K_M) AND (alg.AObs) //Переход: Переход К-М->АОбс
	OR (mde.M_K) AND (alg.AObs) //Переход: Переход М-К->АОбс
					THEN mde.number := enum_mode.AObs;
ELSIF
	   (mde.NObs) AND (btn.NOss.out) //Переход: НОбс->НОсс
	OR (mde.K) AND (btn.NOss.out) //Переход: Кольцо->НОсс
	OR (mde.M) AND (btn.NOss.out) //Переход: Магистраль->НОсс
	OR (mde.K_M) AND (btn.NOss.out) //Переход: Переход К-М->НОсс
	OR (mde.M_K) AND (btn.NOss.out) //Переход: Переход М-К->НОсс
					THEN mde.number := enum_mode.NOss;
ELSIF
	   (mde.K) AND (btn.NObs.out) //Переход: Кольцо->НОбс
	OR (mde.M) AND (btn.NObs.out) //Переход: Магистраль->НОбс
	OR (mde.K_M) AND (btn.NObs.out) //Переход: Переход К-М->НОбс
	OR (mde.M_K) AND (btn.NObs.out) //Переход: Переход М-К->НОбс
					THEN mde.number := enum_mode.NObs;
ELSIF
	   (mde.AOss) AND (AOss.finish AND btn.Unlock.out) //Переход: АОсс->Ремонт
	OR (mde.AObs) AND (AObs.finish AND btn.Unlock.out) //Переход: АОбс->Ремонт
	OR (mde.NOss) AND (NOT ppu.HR AND NOss.finish) //Переход: НОсс->Ремонт
	OR (mde.NObs) AND (NOT ppu.HR AND NObs.finish) //Переход: НОбс->Ремонт
	OR (mde.HR) AND (NOT ppu.HR AND NOT tch.Check_SAU.value OR btn.Repair.out) //Переход: ХР->Ремонт
	OR (mde.GR) AND (NOT ppu.HR AND NOT tch.Check_SAU.value OR btn.Repair.out) //Переход: ГР->Ремонт
	OR (mde.PZ) AND (NOT ppu.HR AND (btn.Cancel.out)) //Переход: ПЗ->Ремонт
	OR (mde.HP) AND (NOT ppu.HR AND HP.finish) //Переход: ХП->Ремонт
	OR (mde.KPK) AND (NOT ppu.HR AND KPK.finish) //Переход: КПК->Ремонт
	OR (mde.Error) AND (TRUE) //Переход: …->Ремонт
					THEN mde.number := enum_mode.Repair;
ELSIF
	   (mde.NOss) AND (ppu.HR AND NOss.finish) //Переход: НОсс->ХР
	OR (mde.NObs) AND (NOT ppu.GR AND ppu.HR AND NObs.finish) //Переход: НОбс->ХР
	OR (mde.Repair) AND (ppu.HR AND ppu.Check_HR.value) //Переход: Ремонт->ХР
	OR (mde.GR) AND (ppu.HR AND NOT ppu.GR AND NOT tch.Check_SAU.value OR btn.HR.out) //Переход: ГР->ХР
	OR (mde.PZ) AND (NOT ppu.GR AND ppu.HR AND (btn.Cancel.out)) //Переход: ПЗ->ХР
	OR (mde.HP) AND (NOT ppu.GR AND ppu.HR AND HP.finish) //Переход: ХП->ХР
	OR (mde.KPK) AND (NOT ppu.GR AND ppu.HR AND KPK.finish) //Переход: КПК->ХР
					THEN mde.number := enum_mode.HR;
ELSIF
	   (mde.NObs) AND (ppu.GR AND ppu.HR AND NObs.finish) //Переход: НОбс->ГР
	OR (mde.Repair) AND (ppu.GR AND ppu.HR AND ppu.Check_GR.value) //Переход: Ремонт->ГР
	OR (mde.HR) AND (ppu.GR AND ppu.HR AND ppu.Check_GR.value) //Переход: ХР->ГР
	OR (mde.PZ) AND (ppu.GR AND ppu.HR AND (btn.Cancel.out)) //Переход: ПЗ->ГР
	OR (mde.HP) AND (ppu.GR AND ppu.HR AND HP.finish) //Переход: ХП->ГР
	OR (mde.KPK) AND (ppu.GR AND ppu.HR AND KPK.finish) //Переход: КПК->ГР
					THEN mde.number := enum_mode.GR;
ELSIF
	   (mde.GR) AND (btn.Start.out AND tch.ReadyPZ.value) //Переход: ГР->ПЗ
					THEN mde.number := enum_mode.PZ;
ELSIF
	   (mde.GR) AND (btn.Start.out AND tch.ReadyHP.value) //Переход: ГР->ХП
					THEN mde.number := enum_mode.HP;
ELSIF
	   (mde.GR) AND (btn.Start.out AND tch.ReadyKPK.value) //Переход: ГР->КПК
					THEN mde.number := enum_mode.KPK;
ELSIF
	   (mde.GR) AND (btn.Start.out AND tch.ReadyAPK.value) //Переход: ГР->АПК
					THEN mde.number := enum_mode.APK;
ELSIF
	   (mde.APK) AND (APK.finish) //Переход: АПК->Кольцо
	OR (mde.M_K) AND (M_K.finish) //Переход: Переход М-К->Кольцо
					THEN mde.number := enum_mode.K;
ELSIF
	   (mde.K_M) AND (K_M.finish) //Переход: Переход К-М->Магистраль
					THEN mde.number := enum_mode.M;
ELSIF
	   (mde.K) AND (btn.K_M.out) //Переход: Кольцо->Переход К-М
	OR (mde.M_K) AND (btn.K_M.out) //Переход: Переход М-К->Переход К-М
					THEN mde.number := enum_mode.K_M;
ELSIF
	   (mde.M) AND (btn.M_K.out) //Переход: Магистраль->Переход М-К
	OR (mde.K_M) AND (btn.M_K.out) //Переход: Переход К-М->Переход М-К
					THEN mde.number := enum_mode.M_K;
END_IF;

//------------------------------------------------------------//
mde.AOss := mde.number = enum_mode.AOss;
mde.AObs := mde.number = enum_mode.AObs;
mde.NOss := mde.number = enum_mode.NOss;
mde.NObs := mde.number = enum_mode.NObs;
mde.Repair := mde.number = enum_mode.Repair;
mde.HR := mde.number = enum_mode.HR;
mde.GR := mde.number = enum_mode.GR;
mde.PZ := mde.number = enum_mode.PZ;
mde.HP := mde.number = enum_mode.HP;
mde.KPK := mde.number = enum_mode.KPK;
mde.APK := mde.number = enum_mode.APK;
mde.K := mde.number = enum_mode.K;
mde.M := mde.number = enum_mode.M;
mde.K_M := mde.number = enum_mode.K_M;
mde.M_K := mde.number = enum_mode.M_K;
mde.Error := mde.number = enum_mode.Error;
//------------------------------------------------------------//

                  
END_FUNCTION

{region INFO}
(*
 Назначение: Используется для обработки входных аналоговых параметров
 Автор:      /Andrey/ 16.07.2025 17:15:05
 Версия ТЭ5: v00.00.01
 Проект:     KA107
*)
{endregion}
FUNCTION aipar_update : BOOL
VAR_INPUT
	cycle : REAL;
END_VAR
VAR
END_VAR

                    aipar.common.cycle := cycle;

aipar.Ntk_1(mdl_value := MODULE_UCP1_A1_FI1.CH01.FREQUENCY, mdl_invalid := MODULE_UCP1_A1_FI1.CH01.INVALID, mdl_hwError := MODULE_UCP1_A1_FI1.HwError); //Частота вращения ТК канал 1
aipar.Nst_1(mdl_value := MODULE_UCP1_A1_FI1.CH02.FREQUENCY, mdl_invalid := MODULE_UCP1_A1_FI1.CH02.INVALID, mdl_hwError := MODULE_UCP1_A1_FI1.HwError); //Частота вращения СТ канал 1
aipar.Ntk_2(mdl_value := MODULE_UCP1_A1_FI2.CH01.FREQUENCY, mdl_invalid := MODULE_UCP1_A1_FI2.CH01.INVALID, mdl_hwError := MODULE_UCP1_A1_FI2.HwError); //Частота вращения ТК канал 2
aipar.Nst_2(mdl_value := MODULE_UCP1_A1_FI2.CH02.FREQUENCY, mdl_invalid := MODULE_UCP1_A1_FI2.CH02.INVALID, mdl_hwError := MODULE_UCP1_A1_FI2.HwError); //Частота вращения СТ канал 2
aipar.Vstk(mdl_value := MODULE_UCP1_A1_AI1.CH01.VALUE, mdl_status := MODULE_UCP1_A1_AI1.CH01.STATUS, mdl_hwError := MODULE_UCP1_A1_AI1.HwError); //Виброскорость ТК
aipar.Vsst(mdl_value := MODULE_UCP1_A1_AI1.CH02.VALUE, mdl_status := MODULE_UCP1_A1_AI1.CH02.STATUS, mdl_hwError := MODULE_UCP1_A1_AI1.HwError); //Виброскорость СТ
aipar.DG_pos(mdl_value := MODULE_UCP1_A1_AI1.CH03.VALUE, mdl_status := MODULE_UCP1_A1_AI1.CH03.STATUS, mdl_hwError := MODULE_UCP1_A1_AI1.HwError); //Положение топливного клапана дозатора газа
aipar.dPmg(mdl_value := MODULE_UCP1_A1_AI1.CH04.VALUE, mdl_status := MODULE_UCP1_A1_AI1.CH04.STATUS, mdl_hwError := MODULE_UCP1_A1_AI1.HwError); //Перепад давления “масло-газ”
aipar.DG_pos_diag(mdl_value := MODULE_UCP1_A1_AI1.CH08.VALUE, mdl_status := MODULE_UCP1_A1_AI1.CH08.STATUS, mdl_hwError := MODULE_UCP1_A1_AI1.HwError); //диаг. (Сигнал управления положением дозатора газа)
aipar.Pa_out14(mdl_value := MODULE_UCP1_A1_AI2.CH01.VALUE, mdl_status := MODULE_UCP1_A1_AI2.CH01.STATUS, mdl_hwError := MODULE_UCP1_A1_AI2.HwError); //Давление воздуха за 14-й ступенью осевого компрессора
aipar.Pg_inN(mdl_value := MODULE_UCP1_A1_AI2.CH02.VALUE, mdl_status := MODULE_UCP1_A1_AI2.CH02.STATUS, mdl_hwError := MODULE_UCP1_A1_AI2.HwError); //Давление газа на входе Н
aipar.Pg_outN(mdl_value := MODULE_UCP1_A1_AI2.CH03.VALUE, mdl_status := MODULE_UCP1_A1_AI2.CH03.STATUS, mdl_hwError := MODULE_UCP1_A1_AI2.HwError); //Давление газа на выходе Н
aipar.Tg_inN(mdl_value := MODULE_UCP1_A1_AI2.CH04.VALUE, mdl_status := MODULE_UCP1_A1_AI2.CH04.STATUS, mdl_hwError := MODULE_UCP1_A1_AI2.HwError); //Температура газа на входе Н
aipar.Tg_outN(mdl_value := MODULE_UCP1_A1_AI2.CH05.VALUE, mdl_status := MODULE_UCP1_A1_AI2.CH05.STATUS, mdl_hwError := MODULE_UCP1_A1_AI2.HwError); //Температура газа на выходе Н
aipar.dP_conf(mdl_value := MODULE_UCP1_A1_AI2.CH06.VALUE, mdl_status := MODULE_UCP1_A1_AI2.CH06.STATUS, mdl_hwError := MODULE_UCP1_A1_AI2.HwError); //Перепад давления на конфузоре
aipar.Vlaz_BA(mdl_value := MODULE_UCP1_A1_AI3.CH02.VALUE, mdl_status := MODULE_UCP1_A1_AI3.CH02.STATUS, mdl_hwError := MODULE_UCP1_A1_AI3.HwError); //Влажность атмосферного воздуха в блоке автоматики
aipar.Ta_BAdown(mdl_value := MODULE_UCP1_A1_AI3.CH03.VALUE, mdl_status := MODULE_UCP1_A1_AI3.CH03.STATUS, mdl_hwError := MODULE_UCP1_A1_AI3.HwError); //Температура атмосферного воздуха в блоке автоматики, нижняя часть
aipar.Ta_BAup(mdl_value := MODULE_UCP1_A1_AI3.CH04.VALUE, mdl_status := MODULE_UCP1_A1_AI3.CH04.STATUS, mdl_hwError := MODULE_UCP1_A1_AI3.HwError); //Температура атмосферного воздуха в блоке автоматики, верхняя часть
aipar.Ptg_inTRK(mdl_value := MODULE_UCP1_A1_AI3.CH05.VALUE, mdl_status := MODULE_UCP1_A1_AI3.CH05.STATUS, mdl_hwError := MODULE_UCP1_A1_AI3.HwError); //Давление топливного газа перед ТРК
aipar.dPtg_inMD(mdl_value := MODULE_UCP1_A1_AI3.CH06.VALUE, mdl_status := MODULE_UCP1_A1_AI3.CH06.STATUS, mdl_hwError := MODULE_UCP1_A1_AI3.HwError); //Перепад давления топливного газа на мерной шайбе ТГ
aipar.Tcool(mdl_value := MODULE_UCP1_A1_AI4.CH01.VALUE, mdl_status := MODULE_UCP1_A1_AI4.CH01.STATUS, mdl_hwError := MODULE_UCP1_A1_AI4.HwError); //Температура холодного спая
aipar.Tup_N(mdl_value := MODULE_UCP1_A1_AI4.CH02.VALUE, mdl_status := MODULE_UCP1_A1_AI4.CH02.STATUS, mdl_hwError := MODULE_UCP1_A1_AI4.HwError); //Температура упорного подшипника Н
aipar.Tm_inD(mdl_value := MODULE_UCP1_A1_AI4.CH03.VALUE, mdl_status := MODULE_UCP1_A1_AI4.CH03.STATUS, mdl_hwError := MODULE_UCP1_A1_AI4.HwError); //Температура масла на входе двигателя
aipar.Tm_outD(mdl_value := MODULE_UCP1_A1_AI4.CH04.VALUE, mdl_status := MODULE_UCP1_A1_AI4.CH04.STATUS, mdl_hwError := MODULE_UCP1_A1_AI4.HwError); //Температура масла на выходе двигателя
aipar.Tm_MB(mdl_value := MODULE_UCP1_A1_AI4.CH06.VALUE, mdl_status := MODULE_UCP1_A1_AI4.CH06.STATUS, mdl_hwError := MODULE_UCP1_A1_AI4.HwError); //Температура масла в баке Д и Н
aipar.Tm_MBU(mdl_value := MODULE_UCP1_A1_AI4.CH07.VALUE, mdl_status := MODULE_UCP1_A1_AI4.CH07.STATUS, mdl_hwError := MODULE_UCP1_A1_AI4.HwError); //Температура масла в баке уплотнения
aipar.Tm_outAVOM(mdl_value := MODULE_UCP1_A1_AI4.CH08.VALUE, mdl_status := MODULE_UCP1_A1_AI4.CH08.STATUS, mdl_hwError := MODULE_UCP1_A1_AI4.HwError); //Температура масла на выходе АВОМ Д и Н
aipar.Ttg(mdl_value := MODULE_UCP1_A1_AI5.CH02.VALUE, mdl_status := MODULE_UCP1_A1_AI5.CH02.STATUS, mdl_hwError := MODULE_UCP1_A1_AI5.HwError); //Температура топливного газа
aipar.Tm_outAU(mdl_value := MODULE_UCP1_A1_AI5.CH03.VALUE, mdl_status := MODULE_UCP1_A1_AI5.CH03.STATUS, mdl_hwError := MODULE_UCP1_A1_AI5.HwError); //Температура масла на выходе АВОМ уплотнений
aipar.Top_N_1(mdl_value := MODULE_UCP1_A1_AI5.CH05.VALUE, mdl_status := MODULE_UCP1_A1_AI5.CH05.STATUS, mdl_hwError := MODULE_UCP1_A1_AI5.HwError); //Температура опорного подшипника №1 Н
aipar.Top_N_2(mdl_value := MODULE_UCP1_A1_AI5.CH06.VALUE, mdl_status := MODULE_UCP1_A1_AI5.CH06.STATUS, mdl_hwError := MODULE_UCP1_A1_AI5.HwError); //Температура опорного подшипника №2 Н
aipar.Tg_inST_1(mdl_value := MODULE_UCP1_A1_AI6.CH01.VALUE, mdl_status := MODULE_UCP1_A1_AI6.CH01.STATUS, mdl_hwError := MODULE_UCP1_A1_AI6.HwError); //Температура газа на входе СТ 1 канал
aipar.Tg_inST_3(mdl_value := MODULE_UCP1_A1_AI6.CH02.VALUE, mdl_status := MODULE_UCP1_A1_AI6.CH02.STATUS, mdl_hwError := MODULE_UCP1_A1_AI6.HwError); //Температура газа на входе СТ 3 канал
aipar.Tg_inST_5(mdl_value := MODULE_UCP1_A1_AI6.CH03.VALUE, mdl_status := MODULE_UCP1_A1_AI6.CH03.STATUS, mdl_hwError := MODULE_UCP1_A1_AI6.HwError); //Температура газа на входе СТ 5 канал
aipar.Tg_inSK(mdl_value := MODULE_UCP1_A1_AI6.CH05.VALUE, mdl_status := MODULE_UCP1_A1_AI6.CH05.STATUS, mdl_hwError := MODULE_UCP1_A1_AI6.HwError); //Температура перед СК
aipar.Tg_inST_2(mdl_value := MODULE_UCP1_A1_AI7.CH01.VALUE, mdl_status := MODULE_UCP1_A1_AI7.CH01.STATUS, mdl_hwError := MODULE_UCP1_A1_AI7.HwError); //Температура газа на входе СТ 2 канал
aipar.Tg_inST_4(mdl_value := MODULE_UCP1_A1_AI7.CH02.VALUE, mdl_status := MODULE_UCP1_A1_AI7.CH02.STATUS, mdl_hwError := MODULE_UCP1_A1_AI7.HwError); //Температура газа на входе СТ 4 канал
aipar.Tg_inST_6(mdl_value := MODULE_UCP1_A1_AI7.CH03.VALUE, mdl_status := MODULE_UCP1_A1_AI7.CH03.STATUS, mdl_hwError := MODULE_UCP1_A1_AI7.HwError); //Температура газа на входе СТ 6 канал
aipar.Ta_inK(mdl_value := MODULE_UCP1_A1_AI7.CH05.VALUE, mdl_status := MODULE_UCP1_A1_AI7.CH05.STATUS, mdl_hwError := MODULE_UCP1_A1_AI7.HwError); //Температура воздуха на входе осевого компрессора

                  
END_FUNCTION

{region INFO}
(*
 Назначение: Используется для обработки выходных аналоговых параметров
 Автор:      /Andrey/ 16.07.2025 17:15:05
 Версия ТЭ5: v00.00.01
 Проект:     KA107
*)
{endregion}
FUNCTION aopar_update : BOOL
VAR_INPUT
END_VAR
VAR
END_VAR

                    aopar.DG_set(mdl_flt := MODULE_UCP1_A2_AO1.STATUS.8, mdl_hwError := MODULE_UCP1_A2_AO1.HwError, mdl_value => MODULE_UCP1_A2_AO1.CH01); //Управление положением дозатора газа

                  
END_FUNCTION

{region INFO}
(*
 Назначение: Используется для обработки входных дискретных параметров
 Автор:      /Andrey/ 16.07.2025 17:15:05
 Версия ТЭ5: v00.00.01
 Проект:     KA107
*)
{endregion}
FUNCTION dipar_update : BOOL
VAR_INPUT
END_VAR
VAR
END_VAR

                    dipar.AO_BA_ai(mdl_value := MODULE_UCP1_A2_DI1.CH01.VALUE, mdl_flt := MODULE_UCP1_A2_DI1.CH01.STATUS.0 OR MODULE_UCP1_A2_DI1.HwError); //АО от блока автоматики ГПА
dipar.AO_BA(mdl_value := dipar.AO_BA_ai.value, mdl_hwError := dipar.AO_BA_ai.flt, mdl_sc := dipar.AO_BA_ai.sc, mdl_brk := dipar.AO_BA_ai.brk); //АО от блока автоматики ГПА

dipar.Fire_OD_ai(mdl_value := MODULE_UCP1_A2_DI1.CH02.VALUE, mdl_flt := MODULE_UCP1_A2_DI1.CH02.STATUS.0 OR MODULE_UCP1_A2_DI1.HwError); //Пожар ОД
dipar.Fire_OD(mdl_value := dipar.Fire_OD_ai.value, mdl_hwError := dipar.Fire_OD_ai.flt, mdl_sc := dipar.Fire_OD_ai.sc, mdl_brk := dipar.Fire_OD_ai.brk); //Пожар ОД

dipar.Lm_MB_Pn_ai(mdl_value := MODULE_UCP1_A2_DI1.CH05.VALUE, mdl_flt := MODULE_UCP1_A2_DI1.CH05.STATUS.0 OR MODULE_UCP1_A2_DI1.HwError); //Уровень масла в МБД+Н минимальный
dipar.Lm_MB_Pn(mdl_value := dipar.Lm_MB_Pn_ai.value, mdl_hwError := dipar.Lm_MB_Pn_ai.flt, mdl_sc := dipar.Lm_MB_Pn_ai.sc, mdl_brk := dipar.Lm_MB_Pn_ai.brk); //Уровень масла в МБД+Н минимальный

dipar.Lm_MBU_Pn_ai(mdl_value := MODULE_UCP1_A2_DI1.CH06.VALUE, mdl_flt := MODULE_UCP1_A2_DI1.CH06.STATUS.0 OR MODULE_UCP1_A2_DI1.HwError); //Уровень масла в МБУпл. минимальный
dipar.Lm_MBU_Pn(mdl_value := dipar.Lm_MBU_Pn_ai.value, mdl_hwError := dipar.Lm_MBU_Pn_ai.flt, mdl_sc := dipar.Lm_MBU_Pn_ai.sc, mdl_brk := dipar.Lm_MBU_Pn_ai.brk); //Уровень масла в МБУпл. минимальный

dipar.Zagaz_OD_Pv_ai(mdl_value := MODULE_UCP1_A2_DI1.CH07.VALUE, mdl_flt := MODULE_UCP1_A2_DI1.CH07.STATUS.0 OR MODULE_UCP1_A2_DI1.HwError); //Загазованность контейнеров выше нормы
dipar.Zagaz_OD_Pv(mdl_value := dipar.Zagaz_OD_Pv_ai.value, mdl_hwError := dipar.Zagaz_OD_Pv_ai.flt, mdl_sc := dipar.Zagaz_OD_Pv_ai.sc, mdl_brk := dipar.Zagaz_OD_Pv_ai.brk); //Загазованность контейнеров выше нормы

dipar.SurgeD_ai(mdl_value := MODULE_UCP1_A2_DI1.CH09.VALUE, mdl_flt := MODULE_UCP1_A2_DI1.CH09.STATUS.0 OR MODULE_UCP1_A2_DI1.HwError); //Помпаж двигателя
dipar.SurgeD(mdl_value := dipar.SurgeD_ai.value, mdl_hwError := dipar.SurgeD_ai.flt, mdl_sc := dipar.SurgeD_ai.sc, mdl_brk := dipar.SurgeD_ai.brk); //Помпаж двигателя

dipar.Pm_TK_An_ai(mdl_value := MODULE_UCP1_A2_DI1.CH10.VALUE, mdl_flt := MODULE_UCP1_A2_DI1.CH10.STATUS.0 OR MODULE_UCP1_A2_DI1.HwError); //Давление масла смазки ТК аварийная
dipar.Pm_TK_An(mdl_value := dipar.Pm_TK_An_ai.value, mdl_hwError := dipar.Pm_TK_An_ai.flt, mdl_sc := dipar.Pm_TK_An_ai.sc, mdl_brk := dipar.Pm_TK_An_ai.brk); //Давление масла смазки ТК аварийная

dipar.Pm_ST_An_ai(mdl_value := MODULE_UCP1_A2_DI1.CH11.VALUE, mdl_flt := MODULE_UCP1_A2_DI1.CH11.STATUS.0 OR MODULE_UCP1_A2_DI1.HwError); //Давление масла смазки СТ аварийная
dipar.Pm_ST_An(mdl_value := dipar.Pm_ST_An_ai.value, mdl_hwError := dipar.Pm_ST_An_ai.flt, mdl_sc := dipar.Pm_ST_An_ai.sc, mdl_brk := dipar.Pm_ST_An_ai.brk); //Давление масла смазки СТ аварийная

dipar.Pm_N_An_ai(mdl_value := MODULE_UCP1_A2_DI1.CH12.VALUE, mdl_flt := MODULE_UCP1_A2_DI1.CH12.STATUS.0 OR MODULE_UCP1_A2_DI1.HwError); //Давление масла смазки Н аварийная
dipar.Pm_N_An(mdl_value := dipar.Pm_N_An_ai.value, mdl_hwError := dipar.Pm_N_An_ai.flt, mdl_sc := dipar.Pm_N_An_ai.sc, mdl_brk := dipar.Pm_N_An_ai.brk); //Давление масла смазки Н аварийная

dipar.dPmg_An_ai(mdl_value := MODULE_UCP1_A2_DI1.CH13.VALUE, mdl_flt := MODULE_UCP1_A2_DI1.CH13.STATUS.0 OR MODULE_UCP1_A2_DI1.HwError); //Аварийный перепад масло-газ
dipar.dPmg_An(mdl_value := dipar.dPmg_An_ai.value, mdl_hwError := dipar.dPmg_An_ai.flt, mdl_sc := dipar.dPmg_An_ai.sc, mdl_brk := dipar.dPmg_An_ai.brk); //Аварийный перепад масло-газ

dipar.Pm_SAR_An_ai(mdl_value := MODULE_UCP1_A2_DI1.CH14.VALUE, mdl_flt := MODULE_UCP1_A2_DI1.CH14.STATUS.0 OR MODULE_UCP1_A2_DI1.HwError); //Давление масла САР < 1,5 МПа
dipar.Pm_SAR_An(mdl_value := dipar.Pm_SAR_An_ai.value, mdl_hwError := dipar.Pm_SAR_An_ai.flt, mdl_sc := dipar.Pm_SAR_An_ai.sc, mdl_brk := dipar.Pm_SAR_An_ai.brk); //Давление масла САР < 1,5 МПа

dipar.dP_F_Pv_ai(mdl_value := MODULE_UCP1_A2_DI2.CH15.VALUE, mdl_flt := MODULE_UCP1_A2_DI2.CH15.STATUS.0 OR MODULE_UCP1_A2_DI2.HwError); //dP перед форсунками камеры сгорания >10кПа
dipar.dP_F_Pv(mdl_value := dipar.dP_F_Pv_ai.value, mdl_hwError := dipar.dP_F_Pv_ai.flt, mdl_sc := dipar.dP_F_Pv_ai.sc, mdl_brk := dipar.dP_F_Pv_ai.brk); //dP перед форсунками камеры сгорания >10кПа

